REGION Network 24 (SCL): 5261/5263 SSC accumulator pressure LO/HI
   "DB_Alarms"."5261_SSC_PIT_01_Low".fLimit := 840.0;
   "DB_Alarms"."5261_SSC_PIT_01_Low".bEnable := TRUE;

   "DB_Alarms"."5263_SSC_PIT_01_High".fLimit := 1400.0;
   "DB_Alarms"."5263_SSC_PIT_01_High".bEnable := TRUE;
END_REGION

REGION Network 25 (SCL): 5262 SSC seal delta T HI
   "DB_Alarms"."5262_DeltaT_ShaftSealHigh".fLimit := 11.0;
   "DB_Alarms"."5262_DeltaT_ShaftSealHigh".bEnable := TRUE;
END_REGION
END_FUNCTION

FUNCTION_BLOCK "InputWarningHandling"   // FB7, FBD
TITLE = Handle I/O warnings
{ S7_Optimized_Access := 'TRUE' }
AUTHOR : Heaten
VERSION : 0.1
// stored: AutoNumber false, IsIECCheckEnabled false, IsRetainMemResEnabled false, MemoryReserve 100, SetENOAutomatically false, UDAEnableTagReadback false
   VAR
      A1101 { ExternalAccessible := 'False'; ExternalVisible := 'False'; ExternalWritable := 'False'; S7_SetPoint := 'True'} : "fbDigitalAlarm";
      A1121 { ExternalAccessible := 'False'; ExternalVisible := 'False'; ExternalWritable := 'False'; S7_SetPoint := 'True'} : "fbDigitalAlarm";
      A1140 { ExternalAccessible := 'False'; ExternalVisible := 'False'; ExternalWritable := 'False'; S7_SetPoint := 'True'} : "fbDigitalAlarm";
      A1216 { ExternalAccessible := 'False'; ExternalVisible := 'False'; ExternalWritable := 'False'; S7_SetPoint := 'True'} : "fbHMIEvent";
      A1217 { ExternalAccessible := 'False'; ExternalVisible := 'False'; ExternalWritable := 'False'; S7_SetPoint := 'True'} : "fbHMIEvent";
      A1218 { ExternalAccessible := 'False'; ExternalVisible := 'False'; ExternalWritable := 'False'; S7_SetPoint := 'True'} : "fbHMIEvent";
      A1224 { ExternalAccessible := 'False'; ExternalVisible := 'False'; ExternalWritable := 'False'; S7_SetPoint := 'True'} : "fbHMIEvent";
      A1225 { ExternalAccessible := 'False'; ExternalVisible := 'False'; ExternalWritable := 'False'; S7_SetPoint := 'True'} : "fbHMIEvent";
      A1226 { ExternalAccessible := 'False'; ExternalVisible := 'False'; ExternalWritable := 'False'; S7_SetPoint := 'True'} : "fbHMIEvent";
      A1227 { ExternalAccessible := 'False'; ExternalVisible := 'False'; ExternalWritable := 'False'; S7_SetPoint := 'True'} : "fbHMIEvent";
      A1228 { ExternalAccessible := 'False'; ExternalVisible := 'False'; ExternalWritable := 'False'; S7_SetPoint := 'True'} : "fbHMIEvent";
      A1229 { ExternalAccessible := 'False'; ExternalVisible := 'False'; ExternalWritable := 'False'; S7_SetPoint := 'True'} : "fbHMIEvent";
      A1230 { ExternalAccessible := 'False'; ExternalVisible := 'False'; ExternalWritable := 'False'; S7_SetPoint := 'True'} : "fbHMIEvent";
      A1234 { ExternalAccessible := 'False'; ExternalVisible := 'False'; ExternalWritable := 'False'; S7_SetPoint := 'True'} : "fbHMIEvent";
      A1235 { ExternalAccessible := 'False'; ExternalVisible := 'False'; ExternalWritable := 'False'; S7_SetPoint := 'True'} : "fbHMIEvent";
      A1236 { ExternalAccessible := 'False'; ExternalVisible := 'False'; ExternalWritable := 'False'; S7_SetPoint := 'True'} : "fbHMIEvent";
      A1237 { ExternalAccessible := 'False'; ExternalVisible := 'False'; ExternalWritable := 'False'; S7_SetPoint := 'True'} : "fbHMIEvent";
      A1238 { ExternalAccessible := 'False'; ExternalVisible := 'False'; ExternalWritable := 'False'; S7_SetPoint := 'True'} : "fbHMIEvent";
      A1239 { ExternalAccessible := 'False'; ExternalVisible := 'False'; ExternalWritable := 'False'; S7_SetPoint := 'True'} : "fbHMIEvent";
      A1240 { ExternalAccessible := 'False'; ExternalVisible := 'False'; ExternalWritable := 'False'; S7_SetPoint := 'True'} : "fbHMIEvent";
      A1245 { ExternalAccessible := 'False'; ExternalVisible := 'False'; ExternalWritable := 'False'; S7_SetPoint := 'True'} : "fbHMIEvent";
      A1246 { ExternalAccessible := 'False'; ExternalVisible := 'False'; ExternalWritable := 'False'; S7_SetPoint := 'True'} : "fbHMIEvent";
      A1247 { ExternalAccessible := 'False'; ExternalVisible := 'False'; ExternalWritable := 'False'; S7_SetPoint := 'True'} : "fbHMIEvent";
      A1248 { ExternalAccessible := 'False'; ExternalVisible := 'False'; ExternalWritable := 'False'; S7_SetPoint := 'True'} : "fbHMIEvent";
      A1249 { ExternalAccessible := 'False'; ExternalVisible := 'False'; ExternalWritable := 'False'; S7_SetPoint := 'True'} : "fbHMIEvent";
      A1251 { ExternalAccessible := 'False'; ExternalVisible := 'False'; ExternalWritable := 'False'; S7_SetPoint := 'True'} : "fbHMIEvent";
      A1252 { ExternalAccessible := 'False'; ExternalVisible := 'False'; ExternalWritable := 'False'; S7_SetPoint := 'True'} : "fbHMIEvent";
      A1253 { ExternalAccessible := 'False'; ExternalVisible := 'False'; ExternalWritable := 'False'; S7_SetPoint := 'True'} : "fbHMIEvent";
      A1254 { ExternalAccessible := 'False'; ExternalVisible := 'False'; ExternalWritable := 'False'; S7_SetPoint := 'True'} : "fbHMIEvent";
      A1258 { ExternalAccessible := 'False'; ExternalVisible := 'False'; ExternalWritable := 'False'; S7_SetPoint := 'True'} : "fbHMIEvent";
      A1259 { ExternalAccessible := 'False'; ExternalVisible := 'False'; ExternalWritable := 'False'; S7_SetPoint := 'True'} : "fbHMIEvent";
      A1260 { ExternalAccessible := 'False'; ExternalVisible := 'False'; ExternalWritable := 'False'; S7_SetPoint := 'True'} : "fbHMIEvent";
      A1262 { ExternalAccessible := 'False'; ExternalVisible := 'False'; ExternalWritable := 'False'; S7_SetPoint := 'True'} : "fbHMIEvent";
      A1263 { ExternalAccessible := 'False'; ExternalVisible := 'False'; ExternalWritable := 'False'; S7_SetPoint := 'True'} : "fbHMIEvent";
      A1265 { ExternalAccessible := 'False'; ExternalVisible := 'False'; ExternalWritable := 'False'; S7_SetPoint := 'True'} : "fbHMIEvent";
      A1269 { ExternalAccessible := 'False'; ExternalVisible := 'False'; ExternalWritable := 'False'; S7_SetPoint := 'True'} : "fbHMIEvent";
      A1270 { ExternalAccessible := 'False'; ExternalVisible := 'False'; ExternalWritable := 'False'; S7_SetPoint := 'True'} : "fbHMIEvent";
      A1271 { ExternalAccessible := 'False'; ExternalVisible := 'False'; ExternalWritable := 'False'; S7_SetPoint := 'True'} : "fbHMIEvent";
      A1272 { ExternalAccessible := 'False'; ExternalVisible := 'False'; ExternalWritable := 'False'; S7_SetPoint := 'True'} : "fbHMIEvent";
      A1273 { ExternalAccessible := 'False'; ExternalVisible := 'False'; ExternalWritable := 'False'; S7_SetPoint := 'True'} : "fbHMIEvent";
      A1275 { ExternalAccessible := 'False'; ExternalVisible := 'False'; ExternalWritable := 'False'; S7_SetPoint := 'True'} : "fbHMIEvent";
      A1293 { ExternalAccessible := 'False'; ExternalVisible := 'False'; ExternalWritable := 'False'; S7_SetPoint := 'True'} : "fbHMIEvent";
      A1294 { S7_SetPoint := 'True'} : "fbDigitalAlarm";
      A1295 { S7_SetPoint := 'True'} : "fbDigitalAlarm";
      A3401 { ExternalAccessible := 'False'; ExternalVisible := 'False'; ExternalWritable := 'False'; S7_SetPoint := 'True'} : "fbDigitalAlarm";
      A5200 { ExternalAccessible := 'False'; ExternalVisible := 'False'; ExternalWritable := 'False'; S7_SetPoint := 'True'} : "fbHMIEvent";
      A5201 { ExternalAccessible := 'False'; ExternalVisible := 'False'; ExternalWritable := 'False'; S7_SetPoint := 'True'} : "fbHMIEvent";
      A5202 { ExternalAccessible := 'False'; ExternalVisible := 'False'; ExternalWritable := 'False'; S7_SetPoint := 'True'} : "fbHMIEvent";
      A5203 { ExternalAccessible := 'False'; ExternalVisible := 'False'; ExternalWritable := 'False'; S7_SetPoint := 'True'} : "fbDigitalAlarm";
      A5204 { ExternalAccessible := 'False'; ExternalVisible := 'False'; ExternalWritable := 'False'; S7_SetPoint := 'True'} : "fbDigitalAlarm";
      A5206 { ExternalAccessible := 'False'; ExternalVisible := 'False'; ExternalWritable := 'False'; S7_SetPoint := 'True'} : "fbHMIEvent";
      A5256 { ExternalAccessible := 'False'; ExternalVisible := 'False'; ExternalWritable := 'False'; S7_SetPoint := 'True'} : "fbHMIEvent";
   END_VAR
BEGIN

REGION Network 1: 1101
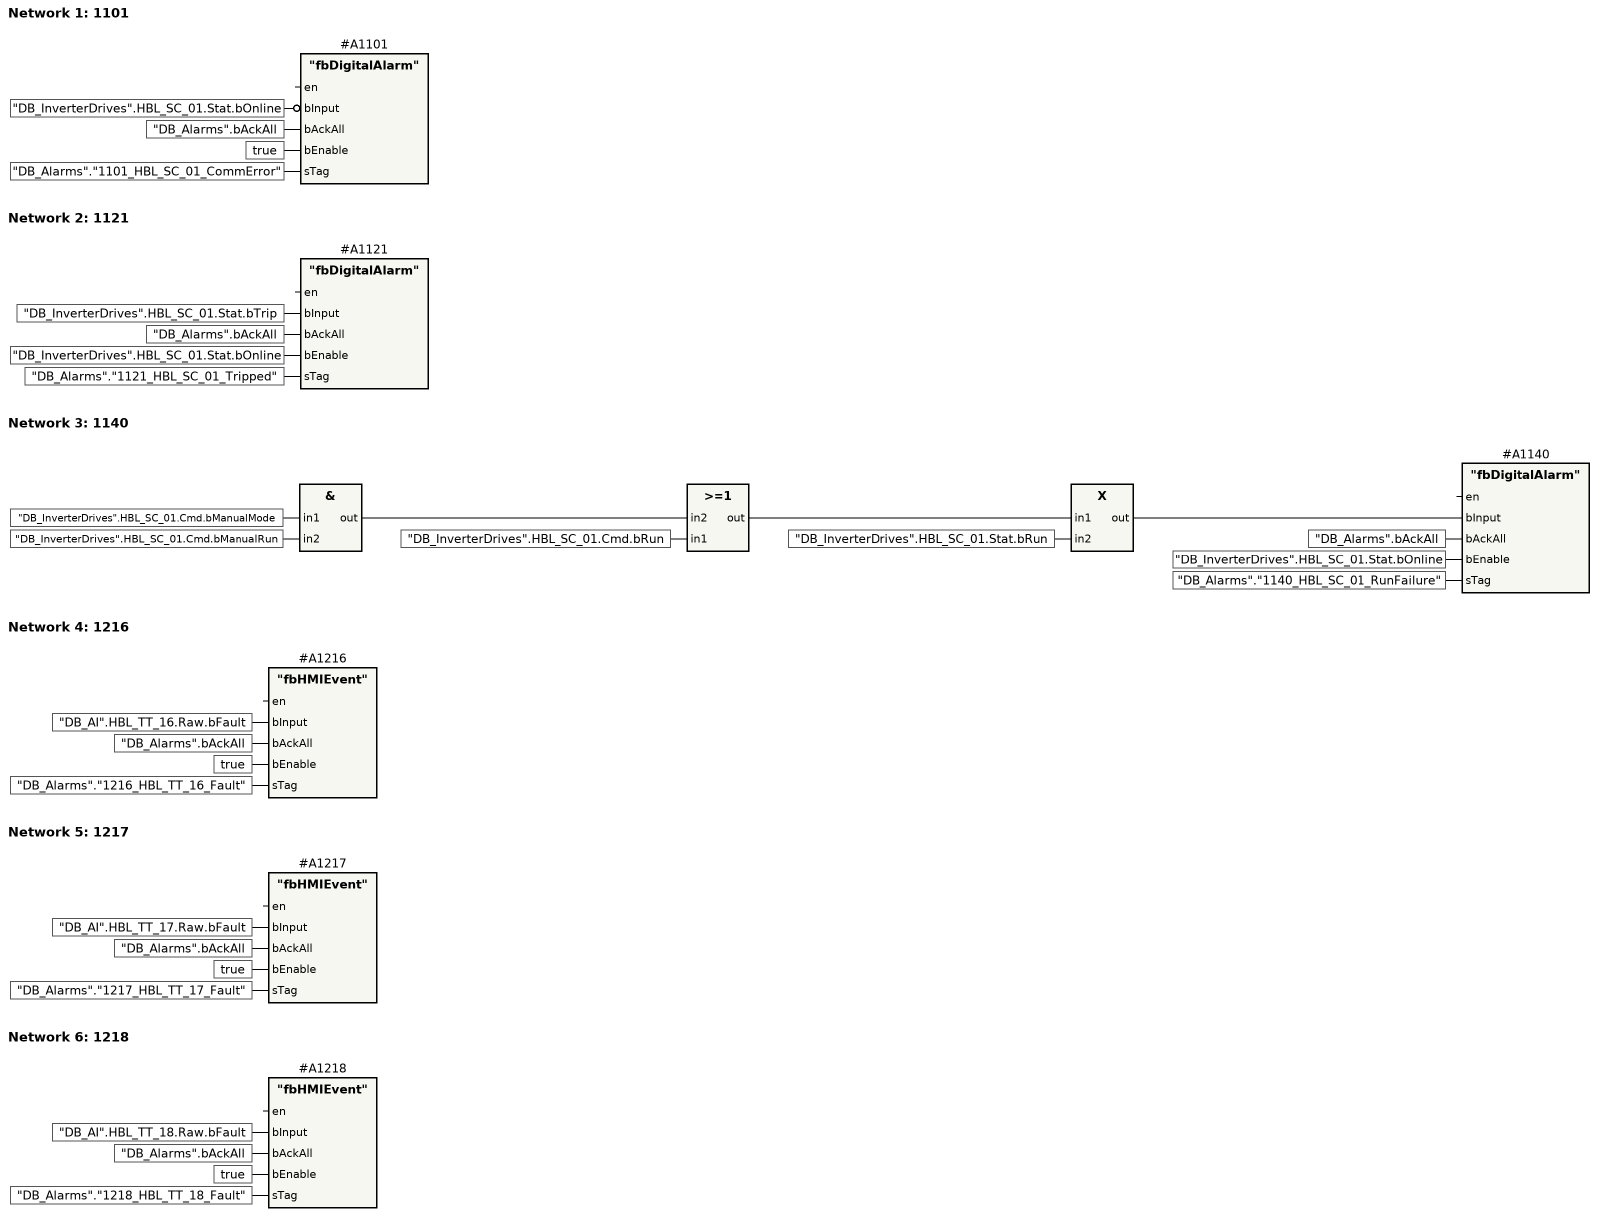
   #A1101(bInput := NOT "DB_InverterDrives".HBL_SC_01.Stat.bOnline,   // "fbDigitalAlarm"
          bAckAll := "DB_Alarms".bAckAll,
          bEnable := true,
          sTag := "DB_Alarms"."1101_HBL_SC_01_CommError");
END_REGION

REGION Network 2: 1121
   #A1121(bInput := "DB_InverterDrives".HBL_SC_01.Stat.bTrip,   // "fbDigitalAlarm"
          bAckAll := "DB_Alarms".bAckAll,
          bEnable := "DB_InverterDrives".HBL_SC_01.Stat.bOnline,
          sTag := "DB_Alarms"."1121_HBL_SC_01_Tripped");
END_REGION

REGION Network 3: 1140
   #A1140(bInput := (("DB_InverterDrives".HBL_SC_01.Cmd.bManualMode AND "DB_InverterDrives".HBL_SC_01.Cmd.bManualRun) OR "DB_InverterDrives".HBL_SC_01.Cmd.bRun) XOR "DB_InverterDrives".HBL_SC_01.Stat.bRun,   // "fbDigitalAlarm"
          bAckAll := "DB_Alarms".bAckAll,
          bEnable := "DB_InverterDrives".HBL_SC_01.Stat.bOnline,
          sTag := "DB_Alarms"."1140_HBL_SC_01_RunFailure");
END_REGION

REGION Network 4: 1216
   #A1216(bInput := "DB_AI".HBL_TT_16.Raw.bFault,   // "fbHMIEvent"
          bAckAll := "DB_Alarms".bAckAll,
          bEnable := true,
          sTag := "DB_Alarms"."1216_HBL_TT_16_Fault");
END_REGION

REGION Network 5: 1217
   #A1217(bInput := "DB_AI".HBL_TT_17.Raw.bFault,   // "fbHMIEvent"
          bAckAll := "DB_Alarms".bAckAll,
          bEnable := true,
          sTag := "DB_Alarms"."1217_HBL_TT_17_Fault");
END_REGION

REGION Network 6: 1218
   #A1218(bInput := "DB_AI".HBL_TT_18.Raw.bFault,   // "fbHMIEvent"
          bAckAll := "DB_Alarms".bAckAll,
          bEnable := true,
          sTag := "DB_Alarms"."1218_HBL_TT_18_Fault");
END_REGION

REGION Network 7: 1224
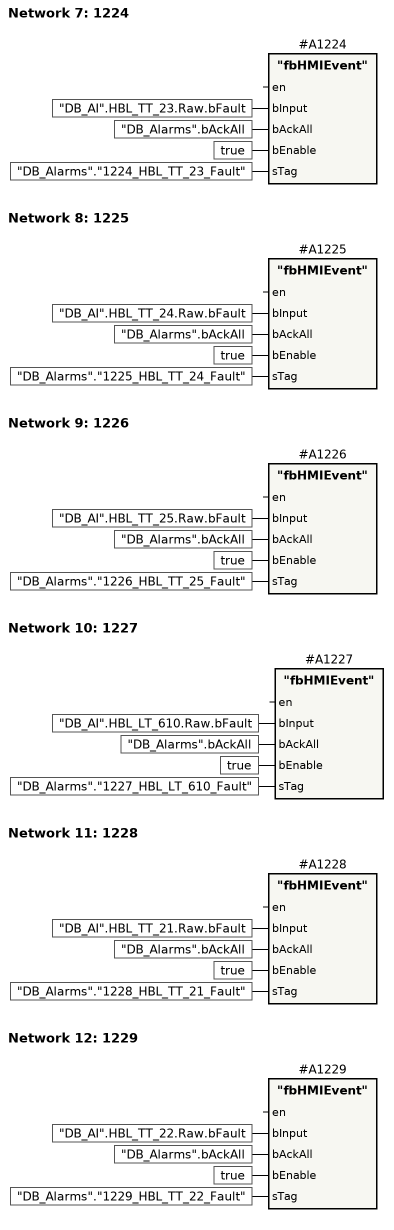
   #A1224(bInput := "DB_AI".HBL_TT_23.Raw.bFault,   // "fbHMIEvent"
          bAckAll := "DB_Alarms".bAckAll,
          bEnable := true,
          sTag := "DB_Alarms"."1224_HBL_TT_23_Fault");
END_REGION

REGION Network 8: 1225
   #A1225(bInput := "DB_AI".HBL_TT_24.Raw.bFault,   // "fbHMIEvent"
          bAckAll := "DB_Alarms".bAckAll,
          bEnable := true,
          sTag := "DB_Alarms"."1225_HBL_TT_24_Fault");
END_REGION

REGION Network 9: 1226
   #A1226(bInput := "DB_AI".HBL_TT_25.Raw.bFault,   // "fbHMIEvent"
          bAckAll := "DB_Alarms".bAckAll,
          bEnable := true,
          sTag := "DB_Alarms"."1226_HBL_TT_25_Fault");
END_REGION

REGION Network 10: 1227
   #A1227(bInput := "DB_AI".HBL_LT_610.Raw.bFault,   // "fbHMIEvent"
          bAckAll := "DB_Alarms".bAckAll,
          bEnable := true,
          sTag := "DB_Alarms"."1227_HBL_LT_610_Fault");
END_REGION

REGION Network 11: 1228
   #A1228(bInput := "DB_AI".HBL_TT_21.Raw.bFault,   // "fbHMIEvent"
          bAckAll := "DB_Alarms".bAckAll,
          bEnable := true,
          sTag := "DB_Alarms"."1228_HBL_TT_21_Fault");
END_REGION

REGION Network 12: 1229
   #A1229(bInput := "DB_AI".HBL_TT_22.Raw.bFault,   // "fbHMIEvent"
          bAckAll := "DB_Alarms".bAckAll,
          bEnable := true,
          sTag := "DB_Alarms"."1229_HBL_TT_22_Fault");
END_REGION

REGION Network 13: 1230
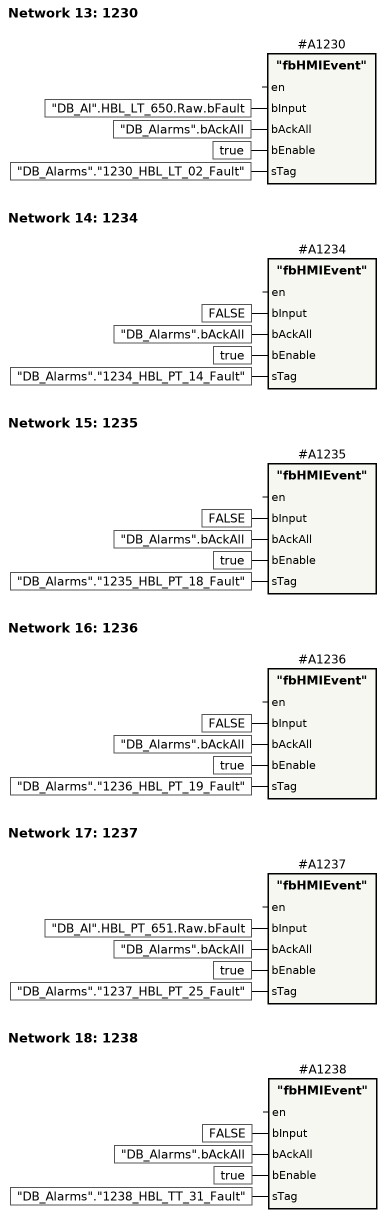
   #A1230(bInput := "DB_AI".HBL_LT_650.Raw.bFault,   // "fbHMIEvent"
          bAckAll := "DB_Alarms".bAckAll,
          bEnable := true,
          sTag := "DB_Alarms"."1230_HBL_LT_02_Fault");
END_REGION

REGION Network 14: 1234
   #A1234(bInput := FALSE,   // "fbHMIEvent"
          bAckAll := "DB_Alarms".bAckAll,
          bEnable := true,
          sTag := "DB_Alarms"."1234_HBL_PT_14_Fault");
END_REGION

REGION Network 15: 1235
   #A1235(bInput := FALSE,   // "fbHMIEvent"
          bAckAll := "DB_Alarms".bAckAll,
          bEnable := true,
          sTag := "DB_Alarms"."1235_HBL_PT_18_Fault");
END_REGION

REGION Network 16: 1236
   #A1236(bInput := FALSE,   // "fbHMIEvent"
          bAckAll := "DB_Alarms".bAckAll,
          bEnable := true,
          sTag := "DB_Alarms"."1236_HBL_PT_19_Fault");
END_REGION

REGION Network 17: 1237
   #A1237(bInput := "DB_AI".HBL_PT_651.Raw.bFault,   // "fbHMIEvent"
          bAckAll := "DB_Alarms".bAckAll,
          bEnable := true,
          sTag := "DB_Alarms"."1237_HBL_PT_25_Fault");
END_REGION

REGION Network 18: 1238
   #A1238(bInput := FALSE,   // "fbHMIEvent"
          bAckAll := "DB_Alarms".bAckAll,
          bEnable := true,
          sTag := "DB_Alarms"."1238_HBL_TT_31_Fault");
END_REGION

REGION Network 19: 1239
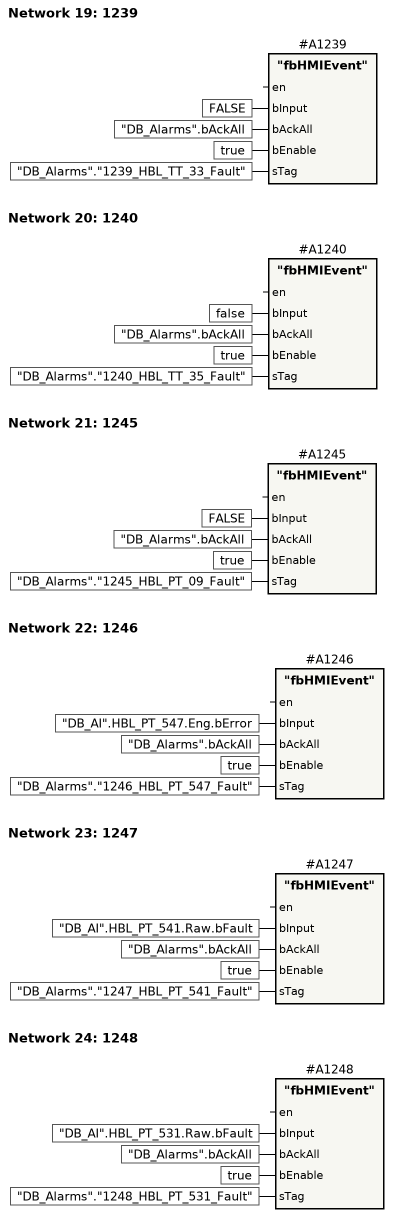
   #A1239(bInput := FALSE,   // "fbHMIEvent"
          bAckAll := "DB_Alarms".bAckAll,
          bEnable := true,
          sTag := "DB_Alarms"."1239_HBL_TT_33_Fault");
END_REGION

REGION Network 20: 1240
   #A1240(bInput := false,   // "fbHMIEvent"
          bAckAll := "DB_Alarms".bAckAll,
          bEnable := true,
          sTag := "DB_Alarms"."1240_HBL_TT_35_Fault");
END_REGION

REGION Network 21: 1245
   #A1245(bInput := FALSE,   // "fbHMIEvent"
          bAckAll := "DB_Alarms".bAckAll,
          bEnable := true,
          sTag := "DB_Alarms"."1245_HBL_PT_09_Fault");
END_REGION

REGION Network 22: 1246
   #A1246(bInput := "DB_AI".HBL_PT_547.Eng.bError,   // "fbHMIEvent"
          bAckAll := "DB_Alarms".bAckAll,
          bEnable := true,
          sTag := "DB_Alarms"."1246_HBL_PT_547_Fault");
END_REGION

REGION Network 23: 1247
   #A1247(bInput := "DB_AI".HBL_PT_541.Raw.bFault,   // "fbHMIEvent"
          bAckAll := "DB_Alarms".bAckAll,
          bEnable := true,
          sTag := "DB_Alarms"."1247_HBL_PT_541_Fault");
END_REGION

REGION Network 24: 1248
   #A1248(bInput := "DB_AI".HBL_PT_531.Raw.bFault,   // "fbHMIEvent"
          bAckAll := "DB_Alarms".bAckAll,
          bEnable := true,
          sTag := "DB_Alarms"."1248_HBL_PT_531_Fault");
END_REGION

REGION Network 25: 1249
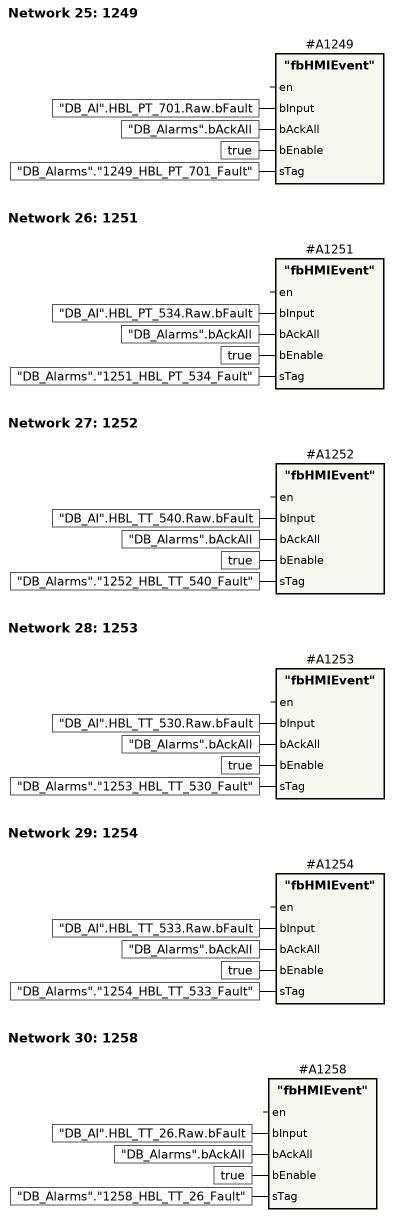
   #A1249(bInput := "DB_AI".HBL_PT_701.Raw.bFault,   // "fbHMIEvent"
          bAckAll := "DB_Alarms".bAckAll,
          bEnable := true,
          sTag := "DB_Alarms"."1249_HBL_PT_701_Fault");
END_REGION

REGION Network 26: 1251
   #A1251(bInput := "DB_AI".HBL_PT_534.Raw.bFault,   // "fbHMIEvent"
          bAckAll := "DB_Alarms".bAckAll,
          bEnable := true,
          sTag := "DB_Alarms"."1251_HBL_PT_534_Fault");
END_REGION

REGION Network 27: 1252
   #A1252(bInput := "DB_AI".HBL_TT_540.Raw.bFault,   // "fbHMIEvent"
          bAckAll := "DB_Alarms".bAckAll,
          bEnable := true,
          sTag := "DB_Alarms"."1252_HBL_TT_540_Fault");
END_REGION

REGION Network 28: 1253
   #A1253(bInput := "DB_AI".HBL_TT_530.Raw.bFault,   // "fbHMIEvent"
          bAckAll := "DB_Alarms".bAckAll,
          bEnable := true,
          sTag := "DB_Alarms"."1253_HBL_TT_530_Fault");
END_REGION

REGION Network 29: 1254
   #A1254(bInput := "DB_AI".HBL_TT_533.Raw.bFault,   // "fbHMIEvent"
          bAckAll := "DB_Alarms".bAckAll,
          bEnable := true,
          sTag := "DB_Alarms"."1254_HBL_TT_533_Fault");
END_REGION

REGION Network 30: 1258
   #A1258(bInput := "DB_AI".HBL_TT_26.Raw.bFault,   // "fbHMIEvent"
          bAckAll := "DB_Alarms".bAckAll,
          bEnable := true,
          sTag := "DB_Alarms"."1258_HBL_TT_26_Fault");
END_REGION

REGION Network 31: 1259
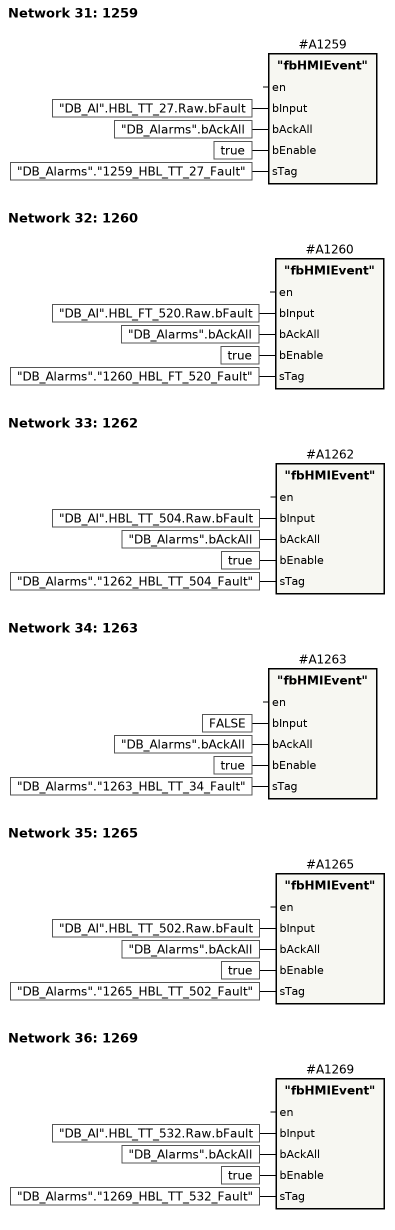
   #A1259(bInput := "DB_AI".HBL_TT_27.Raw.bFault,   // "fbHMIEvent"
          bAckAll := "DB_Alarms".bAckAll,
          bEnable := true,
          sTag := "DB_Alarms"."1259_HBL_TT_27_Fault");
END_REGION

REGION Network 32: 1260
   #A1260(bInput := "DB_AI".HBL_FT_520.Raw.bFault,   // "fbHMIEvent"
          bAckAll := "DB_Alarms".bAckAll,
          bEnable := true,
          sTag := "DB_Alarms"."1260_HBL_FT_520_Fault");
END_REGION

REGION Network 33: 1262
   #A1262(bInput := "DB_AI".HBL_TT_504.Raw.bFault,   // "fbHMIEvent"
          bAckAll := "DB_Alarms".bAckAll,
          bEnable := true,
          sTag := "DB_Alarms"."1262_HBL_TT_504_Fault");
END_REGION

REGION Network 34: 1263
   #A1263(bInput := FALSE,   // "fbHMIEvent"
          bAckAll := "DB_Alarms".bAckAll,
          bEnable := true,
          sTag := "DB_Alarms"."1263_HBL_TT_34_Fault");
END_REGION

REGION Network 35: 1265
   #A1265(bInput := "DB_AI".HBL_TT_502.Raw.bFault,   // "fbHMIEvent"
          bAckAll := "DB_Alarms".bAckAll,
          bEnable := true,
          sTag := "DB_Alarms"."1265_HBL_TT_502_Fault");
END_REGION

REGION Network 36: 1269
   #A1269(bInput := "DB_AI".HBL_TT_532.Raw.bFault,   // "fbHMIEvent"
          bAckAll := "DB_Alarms".bAckAll,
          bEnable := true,
          sTag := "DB_Alarms"."1269_HBL_TT_532_Fault");
END_REGION

REGION Network 37: 1270
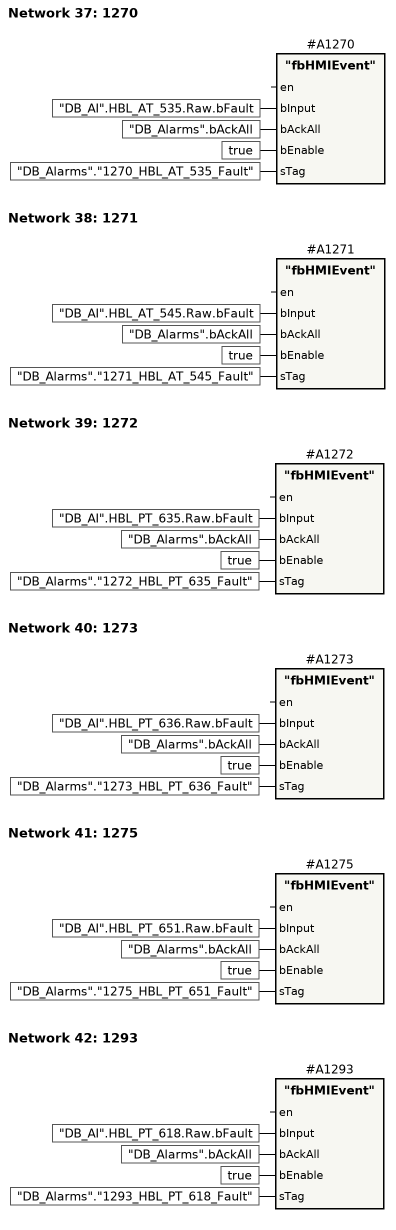
   #A1270(bInput := "DB_AI".HBL_AT_535.Raw.bFault,   // "fbHMIEvent"
          bAckAll := "DB_Alarms".bAckAll,
          bEnable := true,
          sTag := "DB_Alarms"."1270_HBL_AT_535_Fault");
END_REGION

REGION Network 38: 1271
   #A1271(bInput := "DB_AI".HBL_AT_545.Raw.bFault,   // "fbHMIEvent"
          bAckAll := "DB_Alarms".bAckAll,
          bEnable := true,
          sTag := "DB_Alarms"."1271_HBL_AT_545_Fault");
END_REGION

REGION Network 39: 1272
   #A1272(bInput := "DB_AI".HBL_PT_635.Raw.bFault,   // "fbHMIEvent"
          bAckAll := "DB_Alarms".bAckAll,
          bEnable := true,
          sTag := "DB_Alarms"."1272_HBL_PT_635_Fault");
END_REGION

REGION Network 40: 1273
   #A1273(bInput := "DB_AI".HBL_PT_636.Raw.bFault,   // "fbHMIEvent"
          bAckAll := "DB_Alarms".bAckAll,
          bEnable := true,
          sTag := "DB_Alarms"."1273_HBL_PT_636_Fault");
END_REGION

REGION Network 41: 1275
   #A1275(bInput := "DB_AI".HBL_PT_651.Raw.bFault,   // "fbHMIEvent"
          bAckAll := "DB_Alarms".bAckAll,
          bEnable := true,
          sTag := "DB_Alarms"."1275_HBL_PT_651_Fault");
END_REGION

REGION Network 42: 1293
   #A1293(bInput := "DB_AI".HBL_PT_618.Raw.bFault,   // "fbHMIEvent"
          bAckAll := "DB_Alarms".bAckAll,
          bEnable := true,
          sTag := "DB_Alarms"."1293_HBL_PT_618_Fault");
END_REGION

REGION Network 43: 1294
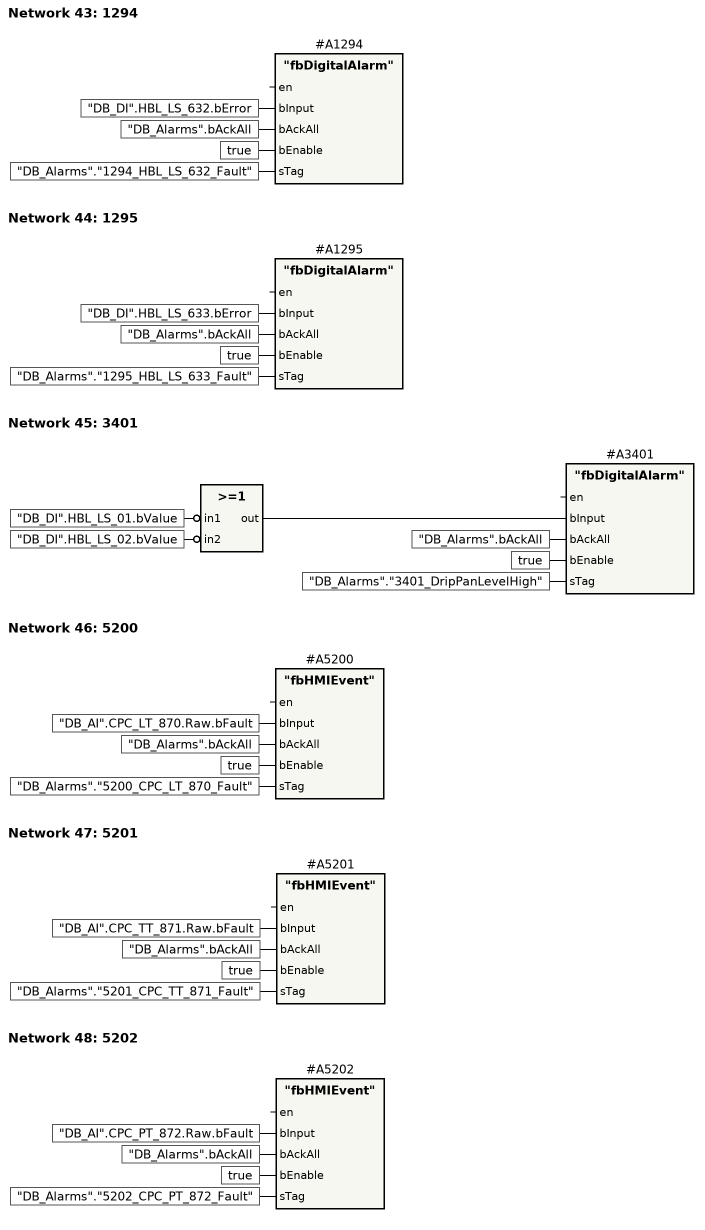
   #A1294(bInput := "DB_DI".HBL_LS_632.bError,   // "fbDigitalAlarm"
          bAckAll := "DB_Alarms".bAckAll,
          bEnable := true,
          sTag := "DB_Alarms"."1294_HBL_LS_632_Fault");
END_REGION

REGION Network 44: 1295
   #A1295(bInput := "DB_DI".HBL_LS_633.bError,   // "fbDigitalAlarm"
          bAckAll := "DB_Alarms".bAckAll,
          bEnable := true,
          sTag := "DB_Alarms"."1295_HBL_LS_633_Fault");
END_REGION

REGION Network 45: 3401
   #A3401(bInput := NOT "DB_DI".HBL_LS_01.bValue OR NOT "DB_DI".HBL_LS_02.bValue,   // "fbDigitalAlarm"
          bAckAll := "DB_Alarms".bAckAll,
          bEnable := true,
          sTag := "DB_Alarms"."3401_DripPanLevelHigh");
END_REGION

REGION Network 46: 5200
   #A5200(bInput := "DB_AI".CPC_LT_870.Raw.bFault,   // "fbHMIEvent"
          bAckAll := "DB_Alarms".bAckAll,
          bEnable := true,
          sTag := "DB_Alarms"."5200_CPC_LT_870_Fault");
END_REGION

REGION Network 47: 5201
   #A5201(bInput := "DB_AI".CPC_TT_871.Raw.bFault,   // "fbHMIEvent"
          bAckAll := "DB_Alarms".bAckAll,
          bEnable := true,
          sTag := "DB_Alarms"."5201_CPC_TT_871_Fault");
END_REGION

REGION Network 48: 5202
   #A5202(bInput := "DB_AI".CPC_PT_872.Raw.bFault,   // "fbHMIEvent"
          bAckAll := "DB_Alarms".bAckAll,
          bEnable := true,
          sTag := "DB_Alarms"."5202_CPC_PT_872_Fault");
END_REGION

REGION Network 49: 5203
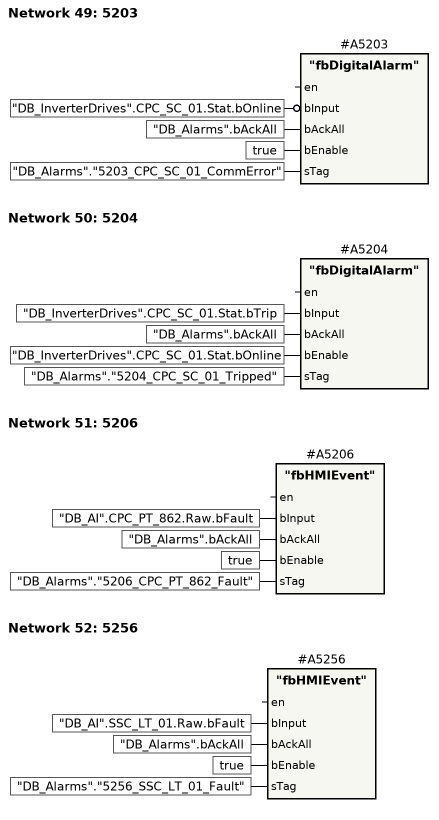
   #A5203(bInput := NOT "DB_InverterDrives".CPC_SC_01.Stat.bOnline,   // "fbDigitalAlarm"
          bAckAll := "DB_Alarms".bAckAll,
          bEnable := true,
          sTag := "DB_Alarms"."5203_CPC_SC_01_CommError");
END_REGION

REGION Network 50: 5204
   // Only show if online
   #A5204(bInput := "DB_InverterDrives".CPC_SC_01.Stat.bTrip,   // "fbDigitalAlarm"
          bAckAll := "DB_Alarms".bAckAll,
          bEnable := "DB_InverterDrives".CPC_SC_01.Stat.bOnline,
          sTag := "DB_Alarms"."5204_CPC_SC_01_Tripped");
END_REGION

REGION Network 51: 5206
   #A5206(bInput := "DB_AI".CPC_PT_862.Raw.bFault,   // "fbHMIEvent"
          bAckAll := "DB_Alarms".bAckAll,
          bEnable := true,
          sTag := "DB_Alarms"."5206_CPC_PT_862_Fault");
END_REGION

REGION Network 52: 5256
   #A5256(bInput := "DB_AI".SSC_LT_01.Raw.bFault,   // "fbHMIEvent"
          bAckAll := "DB_Alarms".bAckAll,
          bEnable := true,
          sTag := "DB_Alarms"."5256_SSC_LT_01_Fault");
END_REGION
END_FUNCTION_BLOCK

FUNCTION_BLOCK "fbDigitalAlarm"   // FB47, FBD
{ S7_Optimized_Access := 'TRUE' }
VERSION : 0.1
// stored: AutoNumber true, IsIECCheckEnabled false, IsRetainMemResEnabled false, MemoryReserve 0, SetENOAutomatically false, UDAEnableTagReadback false
   VAR_INPUT
      bInput : Bool;
      bAckAll : Bool;
      bEnable : Bool;
   END_VAR
   VAR_IN_OUT
      sTag : "stDigitalAlarm";
   END_VAR
   VAR
      Alarm : "fbAlarm";
   END_VAR
BEGIN

REGION Network 1
   // The Enables are ANDed together to allow the struct one to act as a disable bit
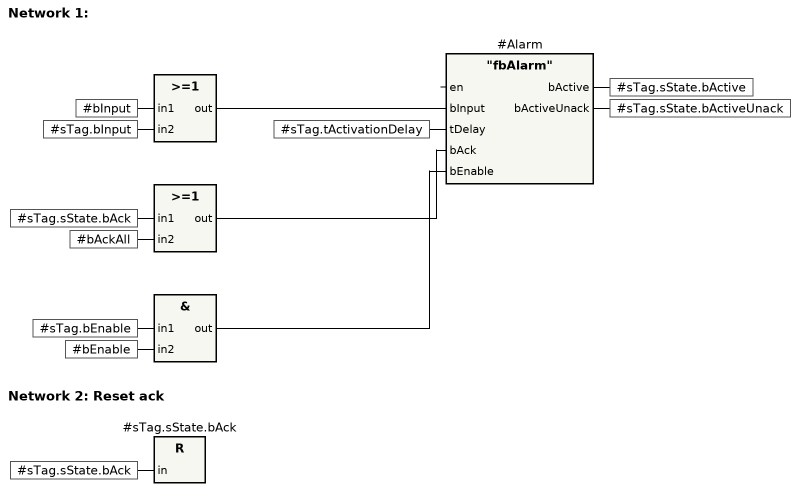
   #Alarm(bInput := #bInput OR #sTag.bInput,   // "fbAlarm"
          tDelay := #sTag.tActivationDelay,
          bAck := #sTag.sState.bAck OR #bAckAll,
          bEnable := #sTag.bEnable AND #bEnable,
          bActive => #sTag.sState.bActive,
          bActiveUnack => #sTag.sState.bActiveUnack);
END_REGION

REGION Network 2: Reset ack
   IF #sTag.sState.bAck THEN #sTag.sState.bAck := FALSE; END_IF;
END_REGION
END_FUNCTION_BLOCK

FUNCTION_BLOCK "fbAlarm"   // FB40, FBD
TITLE = Alarm with time delay
{ S7_Optimized_Access := 'TRUE' }
VERSION : 0.1
// stored: AutoNumber true, IsIECCheckEnabled false, IsRetainMemResEnabled false, MemoryReserve 0, SetENOAutomatically false, UDAEnableTagReadback false
   VAR_INPUT
      bInput : Bool;
      tDelay : Time;
      bAck : Bool;
      bEnable : Bool;
   END_VAR
   VAR_OUTPUT
      bActive : Bool;
      bActiveUnack : Bool;
   END_VAR
   VAR
      DelayTimer : TON_TIME;
      Alarm : Bool;
      AlarmUnack : Bool;
      mActive : Bool;
   END_VAR
   VAR_TEMP
      DelayExpired : Bool;
   END_VAR
   VAR_TEMP   // added for the SCL form of the ladder/FBD networks
      _w1 : Bool;
   END_VAR
BEGIN

REGION Network 1: Delay: alarm must be active for a minimum time period
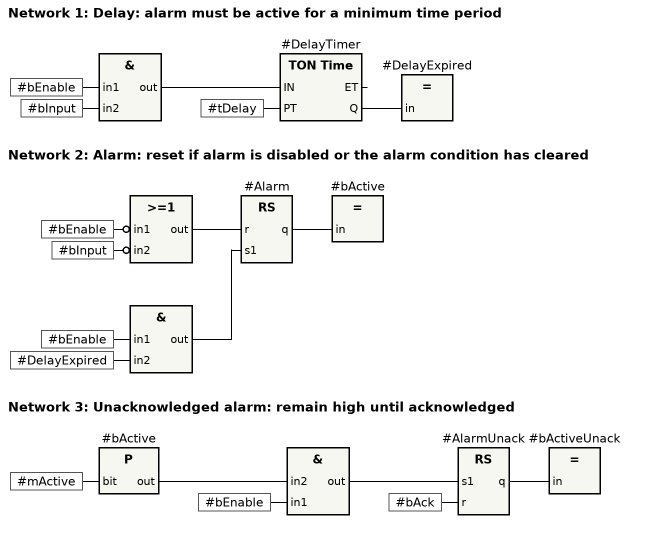
   #DelayTimer(IN := #bEnable AND #bInput, PT := #tDelay);   // TON
   #DelayExpired := #DelayTimer.Q;
END_REGION

REGION Network 2: Alarm: reset if alarm is disabled or the alarm condition has cleared
   IF NOT #bEnable OR NOT #bInput THEN
       #Alarm := FALSE;   // RS flip-flop
   END_IF;
   IF #bEnable AND #DelayExpired THEN #Alarm := TRUE; END_IF;
   #bActive := #Alarm;
END_REGION

REGION Network 3: Unacknowledged alarm: remain high until acknowledged
   #_w1 := #bActive AND NOT #mActive;   // rising edge of #bActive
   #mActive := #bActive;
   IF #bAck THEN
       #AlarmUnack := FALSE;   // RS flip-flop
   END_IF;
   IF #_w1 AND #bEnable THEN #AlarmUnack := TRUE; END_IF;
   #bActiveUnack := #AlarmUnack;
END_REGION
END_FUNCTION_BLOCK

FUNCTION_BLOCK "HMI-Communication"   // FB3, FBD
{ S7_Optimized_Access := 'TRUE' }
VERSION : 0.1
// stored: AutoNumber true, IsIECCheckEnabled false, IsRetainMemResEnabled false, MemoryReserve 0, SetENOAutomatically false, UDAEnableTagReadback false
   VAR
      StartRequest : Bool;
      StopRequest : Bool;
      HMI_Running : Bool;
      SkipPauseTime : Bool;
      EmergencyStopWaitTime : Bool;
      SkipEmergencyStopWait : Bool;
      CloseSafetyRelay : Bool;
      OpenSafetyRelay : Bool;
      HMI_Acknowledge_Error : Bool;
      BackToStandby_OilHeat { ExternalVisible := 'False'; ExternalWritable := 'False'} : Bool;
      BackToStandby_SourceFlowNotOK { ExternalVisible := 'False'; ExternalWritable := 'False'} : Bool;
      BackToStandby_SinkFlowNotOK : Bool;
      BackToStandby_SinkTemperatureNotOK : Bool;
      BackToStandby_SourceTemperatureNotOK : Bool;
      BackToStandby_PerformanceControlNotOK : Bool;
      ReturnValvesManualOverride : Bool;   // Hopefully temporary!
      HBL_XV_02override : Bool;   // Temporary!
      HBL_XV_03override : Bool;   // Temporary!
      HBL_HV_860override : Bool;   // Temporary!
      HBL_HV_861override : Bool;   // Temporary!
      State_Text : String;
      BackToStandby_TriggerBit : Bool;   // Bit set if state changes "back to standby"
      BackToStandby_TriggerMemory : Bool;   // Internal flag memory for "back to standby" changes
      BackToStandby_TriggerInt : Int;   // Integer for state changes "back to standby" HMI message
      BackToStandbyReason_Text : String;   // Text to describe "back to standby" reason
      StopReason_TriggerBit : Bool;
      StopReason_TriggerMemory : Bool;
      StopReason_TriggerInt : Int;
      StopReason_Text : String;
      Progress_Text : Int;
      RegulationTarget : Int;
      RegulationTargetPrev : Int;
      HeatboosterSetpoint : Real;   // Main setpoint of the machine
      HeatboosterSetpointPrev : Real;
      EmergencyStopCountdown : Time_Of_Day;
      A1001 { ExternalAccessible := 'False'; ExternalVisible := 'False'; ExternalWritable := 'False'} : "fbHMIEvent";
      WinCCLink { ExternalAccessible := 'False'; ExternalVisible := 'False'; ExternalWritable := 'False'; S7_SetPoint := 'True'} : "fbHeartbeat";
      State2DwellTimeElapsed { S7_SetPoint := 'True'} : Time_Of_Day;
      State2DwellTime : Time_Of_Day;
      State3DwellTimeElapsed : Time_Of_Day;
      State3DwellTime : Time_Of_Day;
      State4DwellTimeElapsed : Time_Of_Day;
      State4DwellTime : Time_Of_Day;
      State5DwellTimeElapsed : Time_Of_Day;
      State5DwellTime : Time_Of_Day;
      State7DwellTimeElapsed : Time_Of_Day;
      State7DwellTime : Time_Of_Day;
      State2PauseTimeElapsed : Time_Of_Day;
      State2PauseTime : Time_Of_Day;
      PurgeControlPurgeTime : Time_Of_Day;
      PurgeControlSpinTime : Time_Of_Day;
      PerformanceControlStandbyTime : Time_Of_Day;
      PerformanceControlStandbyTimeElapsed : Time_Of_Day;
      FilterDryerOnTime : Time_Of_Day;
      FilterDryerOffTime : Time_Of_Day;
      OilRecoveryOnTime : Time_Of_Day;
      ProgressiveTimes : Array[0..3] of Time_Of_Day;
      ProgressiveTime : Time_Of_Day;
      ProgressiveManualTime : Time_Of_Day;
      HV640_OpenTime : Time_Of_Day;
      HV640_CloseTime : Time_Of_Day;
      HV670_OpenTime : Time_Of_Day;
      HV670_CloseTime : Time_Of_Day;
      HV852_OpenTime : Time_Of_Day;
      HV852_CloseTime : Time_Of_Day;
      HV861_OpenTime : Time_Of_Day;
      HV861_CloseTime : Time_Of_Day;
      State2DwellSync { ExternalAccessible := 'False'; ExternalVisible := 'False'; ExternalWritable := 'False'} : "fbWinCCTime";
      State3DwellSync { ExternalAccessible := 'False'; ExternalVisible := 'False'; ExternalWritable := 'False'; S7_SetPoint := 'True'} : "fbWinCCTime";
      State4DwellSync { ExternalAccessible := 'False'; ExternalVisible := 'False'; ExternalWritable := 'False'; S7_SetPoint := 'True'} : "fbWinCCTime";
      State5DwellSync { ExternalAccessible := 'False'; ExternalVisible := 'False'; ExternalWritable := 'False'; S7_SetPoint := 'True'} : "fbWinCCTime";
      State7DwellSync { ExternalAccessible := 'False'; ExternalVisible := 'False'; ExternalWritable := 'False'; S7_SetPoint := 'True'} : "fbWinCCTime";
      State2PauseSync { ExternalAccessible := 'False'; ExternalVisible := 'False'; ExternalWritable := 'False'; S7_SetPoint := 'True'} : "fbWinCCTime";
      PurgeControlPurgeSync { ExternalAccessible := 'False'; ExternalVisible := 'False'; ExternalWritable := 'False'; S7_SetPoint := 'True'} : "fbWinCCTime";
      PurgeControlSpinSync { ExternalAccessible := 'False'; ExternalVisible := 'False'; ExternalWritable := 'False'; S7_SetPoint := 'True'} : "fbWinCCTime";
      ProgressiveTime0Sync { ExternalAccessible := 'False'; ExternalVisible := 'False'; ExternalWritable := 'False'; S7_SetPoint := 'True'} : "fbWinCCTime";
      ProgressiveTime1Sync { ExternalAccessible := 'False'; ExternalVisible := 'False'; ExternalWritable := 'False'; S7_SetPoint := 'True'} : "fbWinCCTime";
      ProgressiveTime2Sync { ExternalAccessible := 'False'; ExternalVisible := 'False'; ExternalWritable := 'False'; S7_SetPoint := 'True'} : "fbWinCCTime";
      ProgressiveTime3Sync { ExternalAccessible := 'False'; ExternalVisible := 'False'; ExternalWritable := 'False'; S7_SetPoint := 'True'} : "fbWinCCTime";
      ProgressiveManualTimeSync { ExternalAccessible := 'False'; ExternalVisible := 'False'; ExternalWritable := 'False'; S7_SetPoint := 'True'} : "fbWinCCTime";
      PerformanceControlStandbySync { ExternalAccessible := 'False'; ExternalVisible := 'False'; ExternalWritable := 'False'; S7_SetPoint := 'True'} : "fbWinCCTime";
      FilterDryerOnTimeSync { S7_SetPoint := 'True'} : "fbWinCCTime";
      FilterDryerOffTimeSync { S7_SetPoint := 'True'} : "fbWinCCTime";
      OilRecoveryOnTimeSync { S7_SetPoint := 'True'} : "fbWinCCTime";
      HV640_OpenTimeSync { S7_SetPoint := 'True'} : "fbWinCCTime";
      HV640_CloseTimeSync { S7_SetPoint := 'True'} : "fbWinCCTime";
      HV670_OpenTimeSync { S7_SetPoint := 'True'} : "fbWinCCTime";
      HV670_CloseTimeSync { S7_SetPoint := 'True'} : "fbWinCCTime";
      HV852_OpenTimeSync { S7_SetPoint := 'True'} : "fbWinCCTime";
      HV852_CloseTimeSync { S7_SetPoint := 'True'} : "fbWinCCTime";
      HV861_OpenTimeSync { S7_SetPoint := 'True'} : "fbWinCCTime";
      HV861_CloseTimeSync { S7_SetPoint := 'True'} : "fbWinCCTime";
   END_VAR
   VAR_TEMP
      FellBackToStandby_456 : Bool;
      FellBackToStandby_56 : Bool;
   END_VAR
   VAR CONSTANT
      "01_WaitingForStateChange" : SInt := 1;
      "02_ErrorAcknowledge" : SInt := 2;
      "03_SafetyRelayNotClosed" : SInt := 3;
      "04_SafetyRelayInterrupted" : SInt := 4;
      "05_CPU_Init" : SInt := 5;
      "6_CriticalAlarmActive" : SInt := 6;
      "10_ReadyToStart" : SInt := 10;
      "11_EmergencyStopActive" : SInt := 11;
      "12_InverterNotOnline" : SInt := 12;
      "13_ReadyToStartWithActiveWarnings" : SInt := 13;
      "14_EmergencyStopWaitTime" : SInt := 14;
      "20_WaitForSourceFlow" : SInt := 20;
      "21_WaitForSinkFlow" : SInt := 21;
      "22_WaitForSinkHeat" : SInt := 22;
      "23_WaitForSourceHeat" : SInt := 23;
      "24_PauseTime" : SInt := 24;
      "25_PowerControlZeroperformanceDemand" : SInt := 25;
      "26_HeatSink_Limit" : SInt := 26;
      "27_HeatSource_Limit" : SInt := 27;
      "28_VariableControl_Limit" : SInt := 28;
      "29_WaitingForShaftSeal" : SInt := 29;
      "210_State2DwellTime" : Int := 210;
      "30_PerformanceControlNotReady" : SInt := 30;
      "31_LubricationPrimingNotReady" : SInt := 31;
      "39_State3DwellTime" : SInt := 39;
      "50_WaitForOilHeat" : SInt := 50;
      "51_RampingUp" : SInt := 51;
      "52_DryingSuctionLine" : SInt := 52;
      "53_WaitForSuperHeatOut" : SInt := 53;
      "54_WaitForRecuperator" : SInt := 54;
      "55_SuctionManifoldPurge" : SInt := 55;
      "56_StartingAndHydrolock" : SInt := 56;
      "59_State4DwellTime" : SInt := 59;
      "60_Running" : SInt := 60;
      "61_State5DwellTime" : SInt := 61;
      "62_RunningAndHydrolock" : SInt := 62;
      "70_Stopping" : SInt := 70;
      "71_State7DwellTime" : SInt := 71;
      "72_StoppingDrySuctionLine" : SInt := 72;
      "302_PausedInState2" : Int := 302;
      "303_PausedInState3" : Int := 303;
      "304_PausedInState4" : Int := 304;
      "305_PausedInState5" : Int := 305;
      "307_PausedInState7" : Int := 307;
   END_VAR
   VAR_TEMP   // added for the SCL form of the ladder/FBD networks
      _w1 : Bool;
      _w2 : Bool;
   END_VAR
BEGIN

REGION Network 1 (SCL): Comments
   (* 
   What's with the fbWinCCTime & Time_Of_Day variables?

   When WinCC displays a TIME variable, it shows it as an integer number of milliseconds. So 5 minutes is 300,000ms. Not very intutive. 
   For longer times, like 1h20min, it's 4,800,000ms. To get a nice display of HH:MM:SS on the screen, and be able to enter time in this 
   format also, the Time_Of_Day variable type has to be used.

   All regulators & other structs use TIME because it's the right type to use, and the same is used everywhere for uniformity. WinCC 
   requires Time_Of_Day for usability. So instead of wrecking the structure and regularity of all those beautiful structs, a conversion 
   is done here (from TIME to TOD and back) to make TIME values "just work" in WinCC. It's ugly but it works, and frees the structs to be
   made the way the design requires, not the way WinCC requires.
   *)
END_REGION

REGION Network 2: Heartbeat
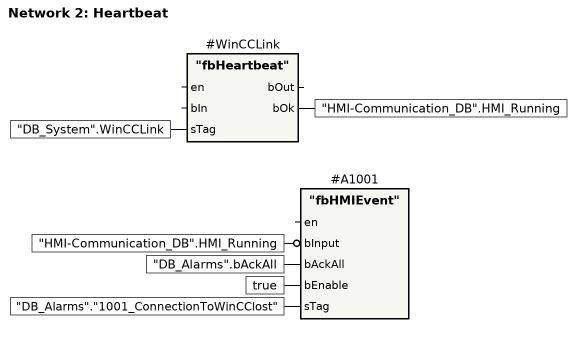
   #WinCCLink(sTag := "DB_System".WinCCLink, bOk => "HMI-Communication_DB".HMI_Running);   // "fbHeartbeat"
   #A1001(bInput := NOT "HMI-Communication_DB".HMI_Running,   // "fbHMIEvent"
          bAckAll := "DB_Alarms".bAckAll,
          bEnable := true,
          sTag := "DB_Alarms"."1001_ConnectionToWinCClost");
END_REGION

REGION Network 3: BackToStandby reason logic
   // Function to show, why the process fell back to standby
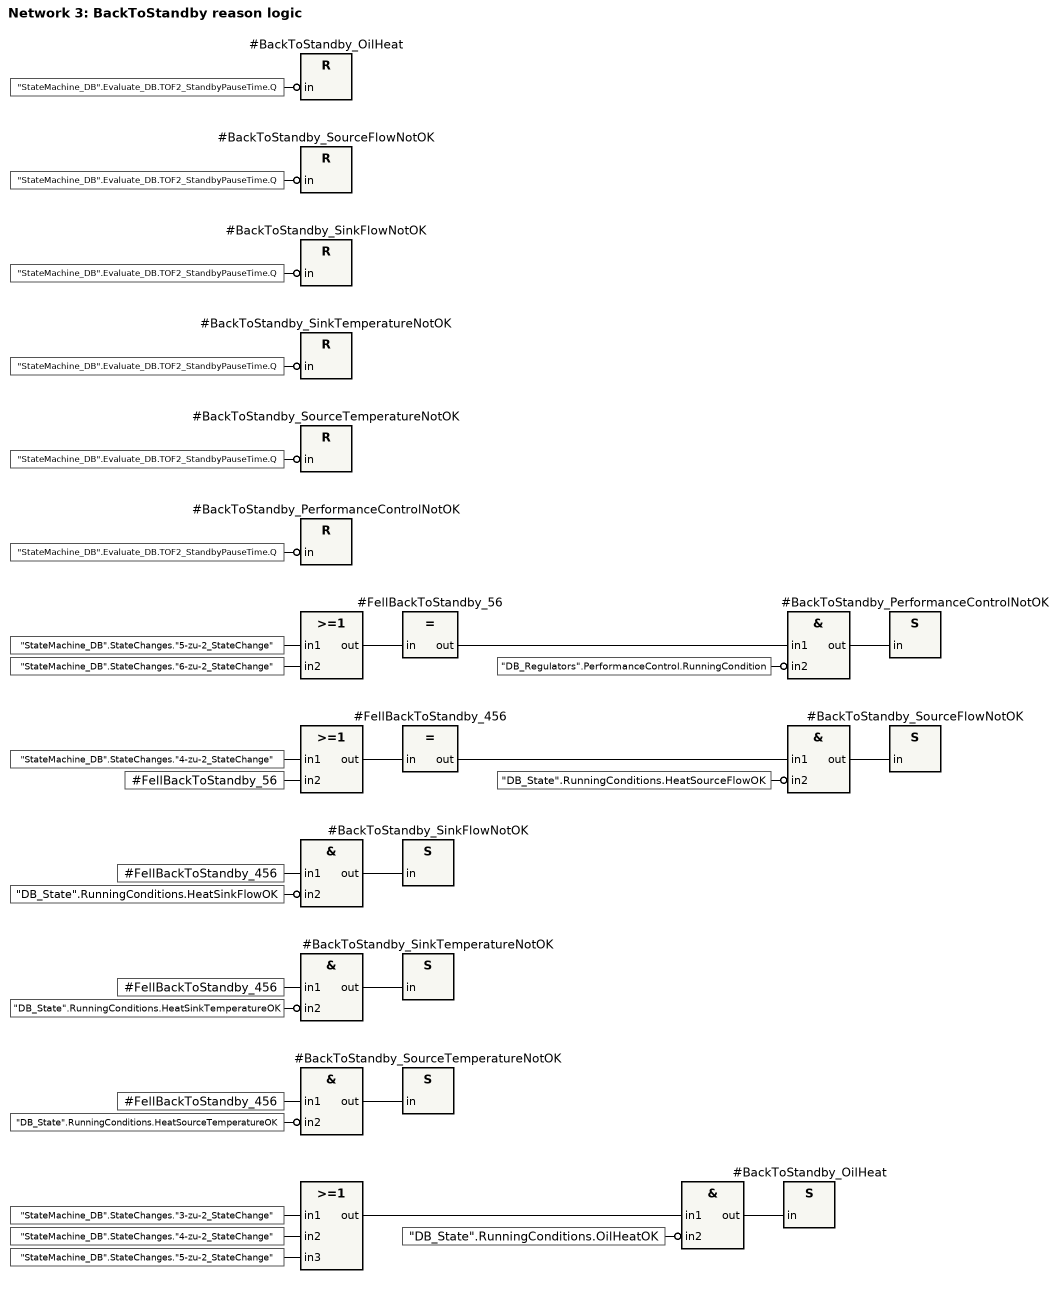
   IF NOT "StateMachine_DB".Evaluate_DB.TOF2_StandbyPauseTime.Q THEN
       #BackToStandby_OilHeat := FALSE;
       #BackToStandby_SourceFlowNotOK := FALSE;
       #BackToStandby_SinkFlowNotOK := FALSE;
       #BackToStandby_SinkTemperatureNotOK := FALSE;
       #BackToStandby_SourceTemperatureNotOK := FALSE;
       #BackToStandby_PerformanceControlNotOK := FALSE;
   END_IF;
   #FellBackToStandby_56 := "StateMachine_DB".StateChanges."5-zu-2_StateChange" OR "StateMachine_DB".StateChanges."6-zu-2_StateChange";
   IF #FellBackToStandby_56 AND NOT "DB_Regulators".PerformanceControl.RunningCondition THEN
       #BackToStandby_PerformanceControlNotOK := TRUE;
   END_IF;
   #FellBackToStandby_456 := "StateMachine_DB".StateChanges."4-zu-2_StateChange" OR #FellBackToStandby_56;
   IF #FellBackToStandby_456 AND NOT "DB_State".RunningConditions.HeatSourceFlowOK THEN
       #BackToStandby_SourceFlowNotOK := TRUE;
   END_IF;
   IF #FellBackToStandby_456 AND NOT "DB_State".RunningConditions.HeatSinkFlowOK THEN
       #BackToStandby_SinkFlowNotOK := TRUE;
   END_IF;
   IF #FellBackToStandby_456 AND NOT "DB_State".RunningConditions.HeatSinkTemperatureOK THEN
       #BackToStandby_SinkTemperatureNotOK := TRUE;
   END_IF;
   IF #FellBackToStandby_456 AND NOT "DB_State".RunningConditions.HeatSourceTemperatureOK THEN
       #BackToStandby_SourceTemperatureNotOK := TRUE;
   END_IF;
   IF ("StateMachine_DB".StateChanges."3-zu-2_StateChange" OR "StateMachine_DB".StateChanges."4-zu-2_StateChange" OR "StateMachine_DB".StateChanges."5-zu-2_StateChange") AND NOT "DB_State".RunningConditions.OilHeatOK THEN
       #BackToStandby_OilHeat := TRUE;
   END_IF;
END_REGION

REGION Network 4: BackToStandby-bit to trigger HMI-Message
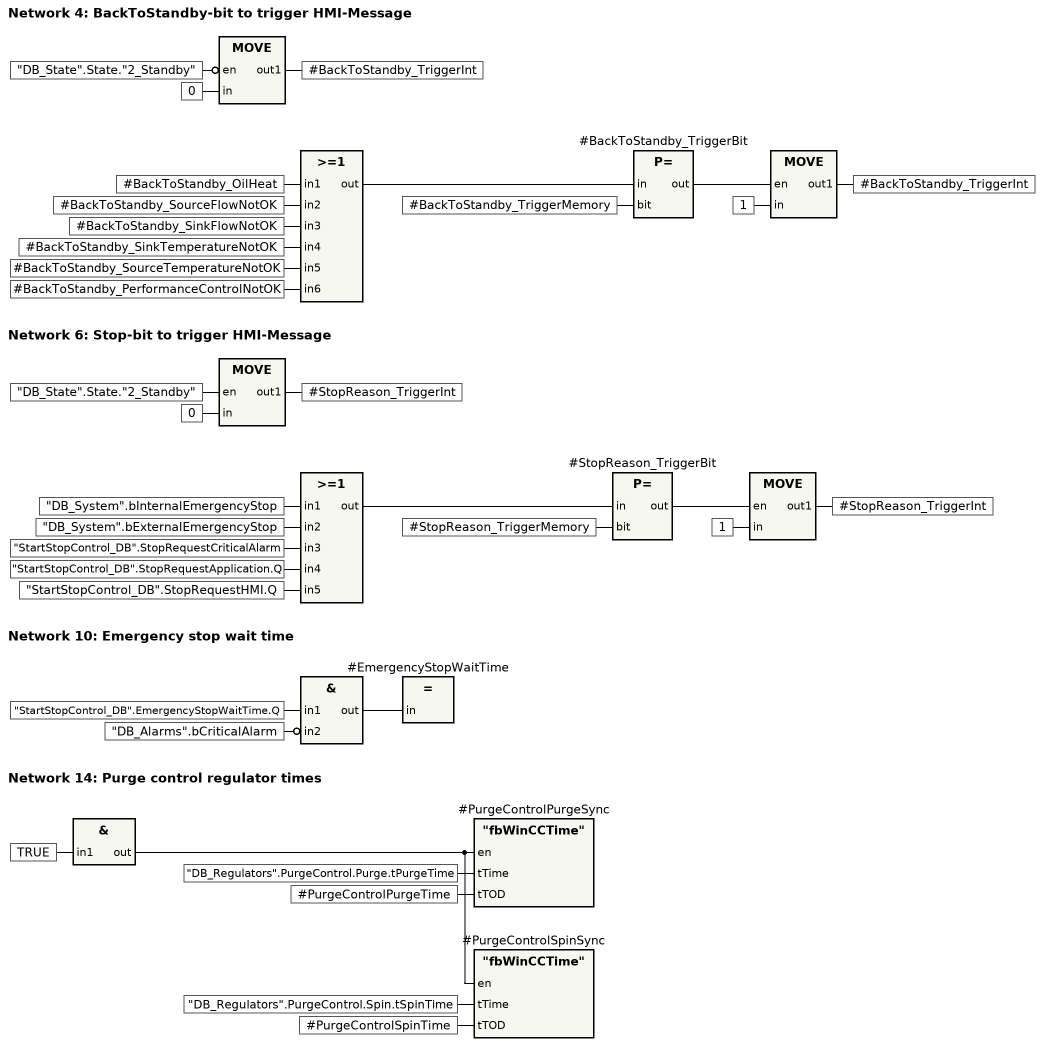
   IF NOT "DB_State".State."2_Standby" THEN #BackToStandby_TriggerInt := 0; END_IF;
   #_w1 := #BackToStandby_OilHeat OR #BackToStandby_SourceFlowNotOK OR #BackToStandby_SinkFlowNotOK OR #BackToStandby_SinkTemperatureNotOK OR #BackToStandby_SourceTemperatureNotOK OR #BackToStandby_PerformanceControlNotOK;
   #BackToStandby_TriggerBit := #_w1 AND NOT #BackToStandby_TriggerMemory;   // rising edge
   #BackToStandby_TriggerMemory := #_w1;
   IF #_w1 THEN #BackToStandby_TriggerInt := 1; END_IF;
END_REGION

REGION Network 5 (SCL): BackToStandby reason text
   // Write "back-to-standby" reason to text and deliver it to the HMI
   IF #BackToStandby_OilHeat THEN
       #BackToStandbyReason_Text := 'Oil heat was not OK!';
   ELSIF #BackToStandby_PerformanceControlNotOK THEN
       #BackToStandbyReason_Text := 'No power was required!';
   ELSIF #BackToStandby_SourceTemperatureNotOK THEN
       #BackToStandbyReason_Text := 'Heat source was not OK!';
   ELSIF #BackToStandby_SinkTemperatureNotOK THEN
       #BackToStandbyReason_Text := 'Heat sink was not OK!';
   ELSIF #BackToStandby_SourceFlowNotOK THEN
       #BackToStandbyReason_Text := 'No source mass flow!';
   ELSIF #BackToStandby_SinkFlowNotOK THEN
       #BackToStandbyReason_Text := 'No sink mass flow!';
   ELSE
       #BackToStandbyReason_Text := '';
   END_IF;
END_REGION

REGION Network 6: Stop-bit to trigger HMI-Message
   IF "DB_State".State."2_Standby" THEN #StopReason_TriggerInt := 0; END_IF;
   #_w1 := "DB_System".bInternalEmergencyStop OR "DB_System".bExternalEmergencyStop OR "StartStopControl_DB".StopRequestCriticalAlarm OR "StartStopControl_DB".StopRequestApplication.Q OR "StartStopControl_DB".StopRequestHMI.Q;
   #StopReason_TriggerBit := #_w1 AND NOT #StopReason_TriggerMemory;   // rising edge
   #StopReason_TriggerMemory := #_w1;
   IF #_w1 THEN #StopReason_TriggerInt := 1; END_IF;
END_REGION

REGION Network 7 (SCL): Stop reason text
   // Write stop reason to text and deliver it to the HMI
   IF "DB_System".bInternalEmergencyStop THEN
       //Emergency Stop intern
       #StopReason_Text := 'Internal emergency stopp!';
   ELSIF "DB_System".bExternalEmergencyStop THEN
       //Emergency Stop extern
       #StopReason_Text := 'External emergency stopp!';
   ELSIF "StartStopControl_DB".StopRequestCriticalAlarm THEN
       //Stop via critical alarm 
       #StopReason_Text := 'Critical alarm!';
   ELSIF "StartStopControl_DB".StopRequestApplication.Q THEN
       //Stop via application PLC
       #StopReason_Text := 'External stopp request!';
   ELSIF "StartStopControl_DB".StopRequestHMI.Q THEN
       //Stop via HMI  
       #StopReason_Text := 'HMI stopp request!';
   END_IF;
END_REGION

REGION Network 8 (SCL): State text & progress text
   // #Progress_Text = 1 is the catch-all error state. If you end up there then there is more work to do.
   CASE "DB_State".State.State_Number OF
       0:  #State_Text := 'Init';

           IF "DB_State".SystemInitialised = FALSE THEN
               #Progress_Text := #"05_CPU_Init";
           ELSE
               #Progress_Text := #"01_WaitingForStateChange";
           END_IF;

       1:  #State_Text := 'Offline';

           IF "DB_System".bEmergencyStop = TRUE THEN
               #Progress_Text := #"11_EmergencyStopActive";
           ELSIF "DB_Alarms"."1110_HBL_SC_10_CommError".sState.bActive OR "DB_Alarms"."1130_HBL_SC_10_Tripped".sState.bActive THEN
               #Progress_Text := #"12_InverterNotOnline";
           ELSIF "DB_Alarms".bCriticalAlarm = TRUE THEN
               #Progress_Text := #"6_CriticalAlarmActive";
           ELSIF "StartStopControl_DB".EmergencyStopWaitTime.Q = TRUE THEN
               #Progress_Text := #"14_EmergencyStopWaitTime";
           ELSIF "DB_Alarms".bCommonAlarm = TRUE THEN
               #Progress_Text := #"13_ReadyToStartWithActiveWarnings";
           ELSE
               #Progress_Text := #"10_ReadyToStart";
           END_IF;


       2:  #State_Text := 'Standby';

           IF "DB_State".RunningConditions.HeatSourceFlowOK = FALSE THEN
               #Progress_Text := #"20_WaitForSourceFlow";
           ELSIF "DB_State".RunningConditions.HeatSinkFlowOK = FALSE THEN
               #Progress_Text := #"21_WaitForSinkFlow";
           ELSIF "DB_State".RunningConditions.HeatSinkTemperatureOK = FALSE THEN
               #Progress_Text := #"22_WaitForSinkHeat";
           ELSIF "DB_State".RunningConditions.HeatSourceTemperatureOK = FALSE THEN
               #Progress_Text := #"23_WaitForSourceHeat";
           ELSIF "StateMachine_DB".Evaluate_DB.TOF2_StandbyPauseTime.Q = TRUE THEN
               #Progress_Text := #"24_PauseTime";
           ELSIF "StateMachine_DB".Evaluate_DB.TON2_Standby.Q = FALSE THEN
               #Progress_Text :=#"210_State2DwellTime";
           ELSIF "DB_Regulators".PerformanceControl.RunningCondition = FALSE THEN
               IF "Regulation_DB".PerformanceControl.HeatSinkTimer.Q = FALSE THEN
                   #Progress_Text := #"26_HeatSink_Limit";
               ELSIF ("Regulation_DB".PerformanceControl.HeatSourceTimer.Q) = FALSE THEN
                   #Progress_Text := #"27_HeatSource_Limit";
               ELSIF "Regulation_DB".PerformanceControl.VariableControlTimer.Q = FALSE THEN
                   #Progress_Text := #"28_VariableControl_Limit";
               ELSE
                   #Progress_Text := #"25_PowerControlZeroperformanceDemand";
               END_IF;
           ELSIF "DB_State".StatePauseFlags[2] = TRUE THEN
               #Progress_Text := #"302_PausedInState2";
           ELSE
               #Progress_Text := #"01_WaitingForStateChange";
           END_IF;

       3:  #State_Text := 'Prepare Start';

           IF "DB_State".RunningConditions.ShaftSealSystemOK = FALSE THEN
               #Progress_Text := #"29_WaitingForShaftSeal";
           ELSIF "DB_State".RunningConditions.OilHeatOK = FALSE THEN
               #Progress_Text := #"50_WaitForOilHeat";
           ELSIF "DB_State".RunningConditions.LubricationPrimingOk = FALSE THEN
               #Progress_Text := #"31_LubricationPrimingNotReady";
           ELSIF "DB_Regulators".PerformanceControl.RunningCondition = FALSE THEN
               #Progress_Text := #"30_PerformanceControlNotReady";
           ELSIF "StateMachine_DB".Evaluate_DB.TON3_PrepareStart.Q = FALSE THEN
               #Progress_Text := #"39_State3DwellTime";
           ELSIF "DB_State".StatePauseFlags[3] = TRUE THEN
               #Progress_Text := #"303_PausedInState3";
           ELSE
               #Progress_Text := #"01_WaitingForStateChange";
           END_IF;

       4:  #State_Text := 'Starting';

           IF "DB_State".RunningConditions.DoWarmStart = FALSE AND "DB_Regulators".PurgeControl.bDone = FALSE THEN
               #Progress_Text := #"55_SuctionManifoldPurge";
           ELSIF "DB_State".RunningConditions.AtOrAboveHydrolockSpeed = FALSE THEN
               #Progress_Text := #"51_RampingUp";
           ELSIF "DB_State".RunningConditions.SuctionLineDry = FALSE THEN
               #Progress_Text := #"52_DryingSuctionLine";
           ELSIF "StateMachine_DB".Evaluate_DB.TON4_Start.Q = FALSE THEN
               #Progress_Text := #"59_State4DwellTime";
           ELSIF "DB_State".StatePauseFlags[4] = TRUE THEN
               #Progress_Text := #"304_PausedInState4";
           ELSE
               #Progress_Text := #"01_WaitingForStateChange";
           END_IF;

       5:  #State_Text := 'Warm-up';

           IF "DB_State".RunningConditions.RiskOfHydrolock = TRUE THEN
               #Progress_Text := #"56_StartingAndHydrolock";
           ELSIF "DB_State".RunningConditions.SuperheatCompressorOutOK = FALSE THEN
               #Progress_Text := #"53_WaitForSuperHeatOut";
           ELSIF "DB_State".RunningConditions.RecuperatorWorking = FALSE THEN
               #Progress_Text := #"54_WaitForRecuperator";
           ELSIF "StateMachine_DB".Evaluate_DB.TON5_Warmup.Q = FALSE THEN
               #Progress_Text := #"61_State5DwellTime";
           ELSIF "DB_State".StatePauseFlags[5] = TRUE THEN
               #Progress_Text := #"305_PausedInState5";
           ELSE
               #Progress_Text := #"01_WaitingForStateChange";
           END_IF;

       6:  #State_Text := 'Running';
           IF "DB_State".RunningConditions.RiskOfHydrolock = TRUE THEN
               #Progress_Text := #"62_RunningAndHydrolock";
           ELSE
               #Progress_Text := #"60_Running";
           END_IF;

       7:  #State_Text := 'Stop';

           IF "DB_State".RunningConditions.SuctionLineDry = FALSE AND"DB_State".FastStop = FALSE THEN
               #Progress_Text := #"72_StoppingDrySuctionLine";
           ELSIF "DB_InverterDrives".HBL_SC_10.Stat.Speed.Eng.fValue <> 0 THEN
               #Progress_Text := #"70_Stopping";
           ELSIF "StateMachine_DB".Evaluate_DB.TON7_Stop.Q = FALSE THEN
               #Progress_Text := #"71_State7DwellTime";
           ELSE
               #Progress_Text := #"01_WaitingForStateChange";
           END_IF;

       ELSE  
           #State_Text := 'No state!';
   END_CASE;
END_REGION

REGION Network 9 (SCL): Regulation target
   // Repeating some of the logic from PerformanceControl (FB9) here, making it fragile
   // Conditions are evaluated as repeated IFs and not ELSIFs because that is how it is evaluated in FB9. Yes, confusing.
   // This network provides an alternative interface to Performance Control, using its public API (DB_Regulators.PerformanceControl)
   // Figure out which target is active & select setpoint
   IF "DB_Regulators".PerformanceControl.Settings.HeatSink.Control_Active THEN
       IF "DB_Regulators".PerformanceControl.Settings.HeatSink.UseFeedFlow THEN
           #RegulationTarget := 2;
       ELSE
           #RegulationTarget := 1;
       END_IF;
   END_IF;

   IF "DB_Regulators".PerformanceControl.Settings.HeatSource.Control_Active THEN
       IF "DB_Regulators".PerformanceControl.Settings.HeatSource.UseFeedFlow THEN
           #RegulationTarget := 4;
       ELSE
           #RegulationTarget := 3;
       END_IF;
   END_IF;

   IF "DB_Regulators".PerformanceControl.Settings.VariableControl.Control_Active AND "DB_Regulators".PerformanceControl.Settings.VariableControl.ReferenceID > 0 THEN
       #RegulationTarget := 6;
   END_IF;

   // Update the currently selected setpoint if updated from HMI
   IF #HeatboosterSetpoint <> #HeatboosterSetpointPrev THEN
       // Select the right setpoint
       CASE #RegulationTarget OF
       1..2 : "DB_Regulators".PerformanceControl.Settings.HeatSink.Setpoint := #HeatboosterSetpoint;
       3..4 : "DB_Regulators".PerformanceControl.Settings.HeatSource.Setpoint := #HeatboosterSetpoint;
       6    : "DB_Regulators".PerformanceControl.Settings.VariableControl.Setpoint := #HeatboosterSetpoint;
       END_CASE;
   END_IF;
   #HeatboosterSetpointPrev := #HeatboosterSetpoint;
END_REGION

REGION Network 10: Emergency stop wait time
   // Do not show when a critical alarm is active
   #EmergencyStopWaitTime := "StartStopControl_DB".EmergencyStopWaitTime.Q AND NOT "DB_Alarms".bCriticalAlarm;
END_REGION

REGION Network 11 (SCL): Emergency lock time
   // Gruesome, this needs refactoring
   #EmergencyStopCountdown := TIME_TO_TOD(IN := ("StartStopControl_DB".EmergencyStopWaitTime.PT - "StartStopControl_DB".EmergencyStopWaitTime.ET));
   IF #SkipEmergencyStopWait THEN
       RESET_TIMER("StartStopControl_DB".EmergencyStopWaitTime);
   END_IF;
END_REGION

REGION Network 12 (SCL): Dwell times
   #State2DwellTimeElapsed := TIME_TO_TOD("StateMachine_DB".Evaluate_DB.TON2_Standby.ET);
   #State2DwellSync(tTime := "DB_CurrentSetting".MissingSetting.Misc.State2DwellTime, tTOD := #State2DwellTime);

   #State3DwellTimeElapsed := TIME_TO_TOD("StateMachine_DB".Evaluate_DB.TON3_PrepareStart.ET);
   #State3DwellSync(tTime := "DB_CurrentSetting".MissingSetting.Misc.State3DwellTime, tTOD := #State3DwellTime);

   #State4DwellTimeElapsed := TIME_TO_TOD("StateMachine_DB".Evaluate_DB.TON4_Start.ET);
   #State4DwellSync(tTime := "DB_CurrentSetting".MissingSetting.Misc.State4DwellTime, tTOD := #State4DwellTime);

   #State5DwellTimeElapsed := TIME_TO_TOD("StateMachine_DB".Evaluate_DB.TON5_Warmup.ET);
   #State5DwellSync(tTime := "DB_CurrentSetting".MissingSetting.Misc.State5DwellTime, tTOD := #State5DwellTime);

   #State7DwellTimeElapsed := TIME_TO_TOD("StateMachine_DB".Evaluate_DB.TON7_Stop.ET);
   #State7DwellSync(tTime := "DB_CurrentSetting".MissingSetting.Misc.State7DwellTime, tTOD := #State7DwellTime);
END_REGION

REGION Network 13 (SCL): Pause time
   #State2PauseTimeElapsed := TIME_TO_TOD("StateMachine_DB".Evaluate_DB.TOF2_StandbyPauseTime.ET);
   #State2PauseSync(tTime := "DB_CurrentSetting".MissingSetting.Misc.State2PauseTime, tTOD := #State2PauseTime);
END_REGION

REGION Network 14: Purge control regulator times
   IF TRUE THEN
       #PurgeControlPurgeSync(tTime := "DB_Regulators".PurgeControl.Purge.tPurgeTime,   // "fbWinCCTime"
                              tTOD := #PurgeControlPurgeTime);
       #PurgeControlSpinSync(tTime := "DB_Regulators".PurgeControl.Spin.tSpinTime, tTOD := #PurgeControlSpinTime);   // "fbWinCCTime"
   END_IF;
END_REGION

REGION Network 15: CPC progressive regulator
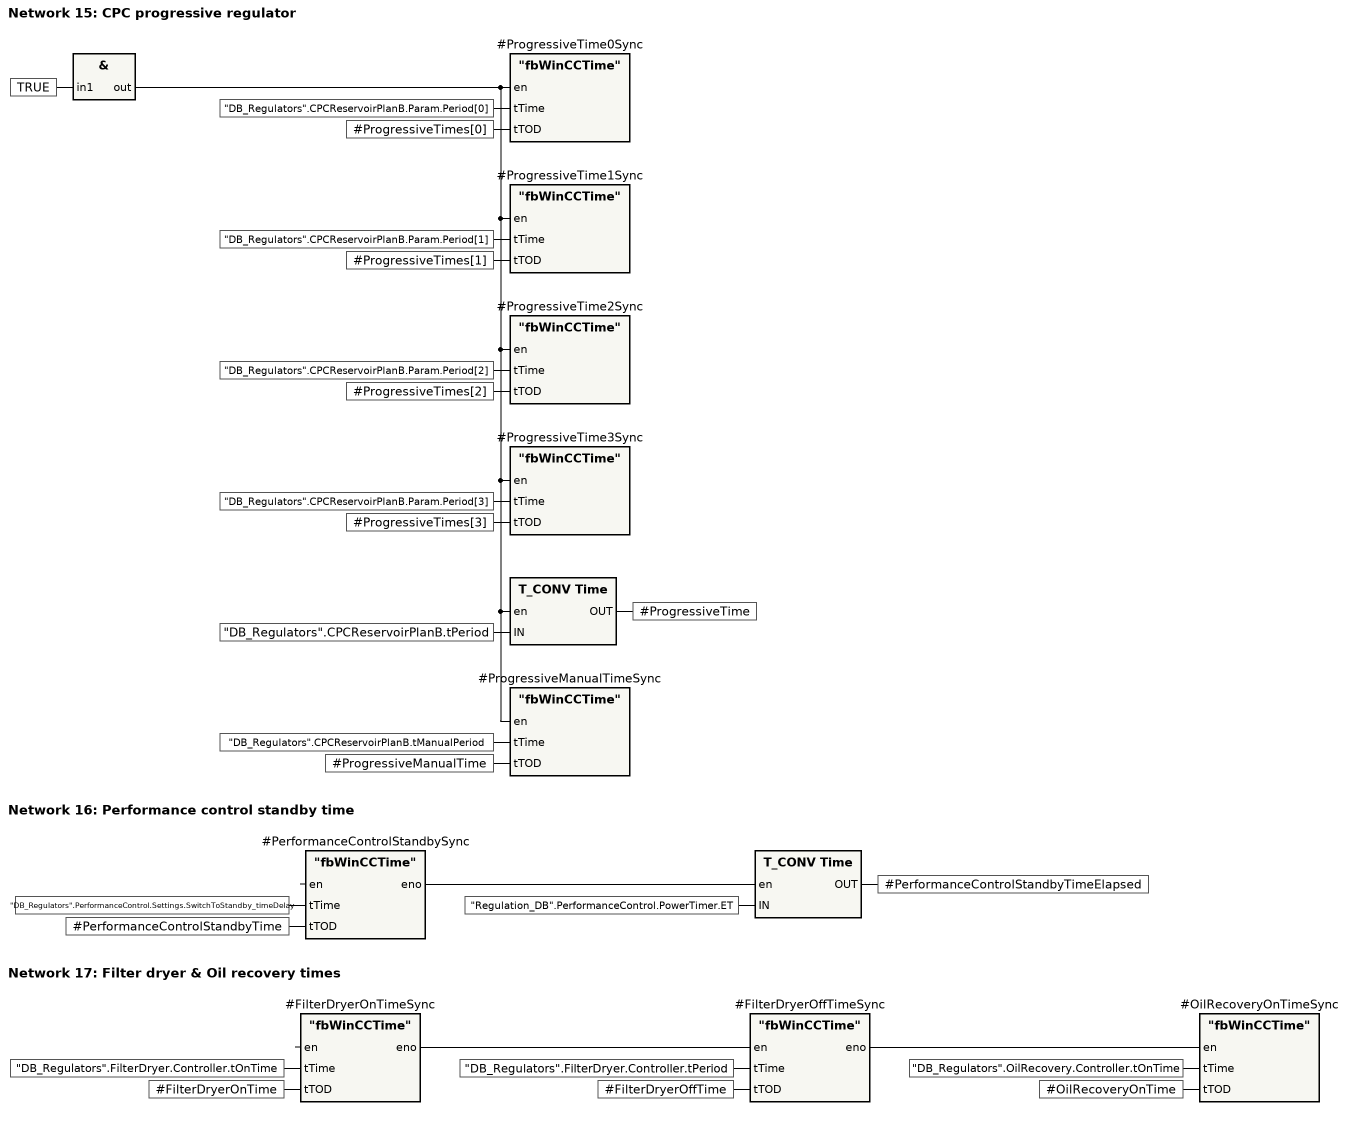
   IF TRUE THEN
       #ProgressiveTime0Sync(tTime := "DB_Regulators".CPCReservoirPlanB.Param.Period[0],   // "fbWinCCTime"
                             tTOD := #ProgressiveTimes[0]);
       #ProgressiveTime1Sync(tTime := "DB_Regulators".CPCReservoirPlanB.Param.Period[1],   // "fbWinCCTime"
                             tTOD := #ProgressiveTimes[1]);
       #ProgressiveTime2Sync(tTime := "DB_Regulators".CPCReservoirPlanB.Param.Period[2],   // "fbWinCCTime"
                             tTOD := #ProgressiveTimes[2]);
       #ProgressiveTime3Sync(tTime := "DB_Regulators".CPCReservoirPlanB.Param.Period[3],   // "fbWinCCTime"
                             tTOD := #ProgressiveTimes[3]);
       T_CONV(IN := "DB_Regulators".CPCReservoirPlanB.tPeriod, OUT => #ProgressiveTime);
       #ProgressiveManualTimeSync(tTime := "DB_Regulators".CPCReservoirPlanB.tManualPeriod,   // "fbWinCCTime"
                               tTOD := #ProgressiveManualTime);
   END_IF;
END_REGION

REGION Network 16: Performance control standby time
   #PerformanceControlStandbySync(tTime := "DB_Regulators".PerformanceControl.Settings.SwitchToStandby_timeDelay,   // "fbWinCCTime"
                           tTOD := #PerformanceControlStandbyTime,
                           ENO => #_w1);
   IF #_w1 THEN
       T_CONV(IN := "Regulation_DB".PerformanceControl.PowerTimer.ET, OUT => #PerformanceControlStandbyTimeElapsed);
   END_IF;
END_REGION

REGION Network 17: Filter dryer & Oil recovery times
   #FilterDryerOnTimeSync(tTime := "DB_Regulators".FilterDryer.Controller.tOnTime,   // "fbWinCCTime"
                          tTOD := #FilterDryerOnTime,
                          ENO => #_w1);
   #FilterDryerOffTimeSync(EN := #_w1,   // "fbWinCCTime"
                           tTime := "DB_Regulators".FilterDryer.Controller.tPeriod,
                           tTOD := #FilterDryerOffTime,
                           ENO => #_w2);
   IF #_w2 THEN
       #OilRecoveryOnTimeSync(tTime := "DB_Regulators".OilRecovery.Controller.tOnTime, tTOD := #OilRecoveryOnTime);   // "fbWinCCTime"
   END_IF;
END_REGION

REGION Network 18: Process Valves
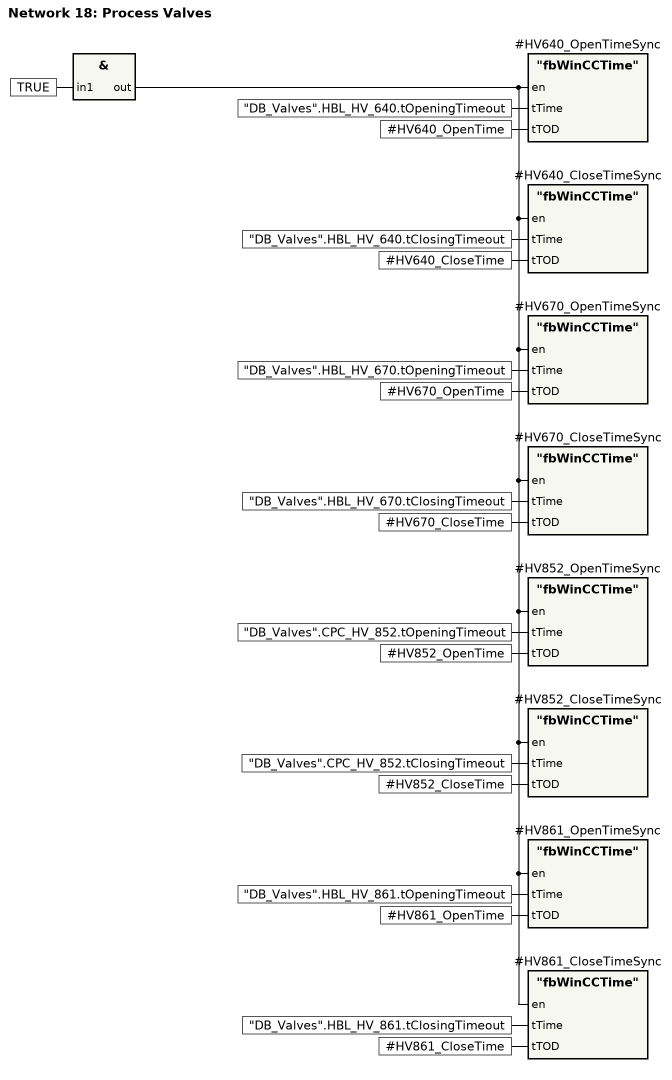
   IF TRUE THEN
       #HV640_OpenTimeSync(tTime := "DB_Valves".HBL_HV_640.tOpeningTimeout, tTOD := #HV640_OpenTime);   // "fbWinCCTime"
       #HV640_CloseTimeSync(tTime := "DB_Valves".HBL_HV_640.tClosingTimeout, tTOD := #HV640_CloseTime);   // "fbWinCCTime"
       #HV670_OpenTimeSync(tTime := "DB_Valves".HBL_HV_670.tOpeningTimeout, tTOD := #HV670_OpenTime);   // "fbWinCCTime"
       #HV670_CloseTimeSync(tTime := "DB_Valves".HBL_HV_670.tClosingTimeout, tTOD := #HV670_CloseTime);   // "fbWinCCTime"
       #HV852_OpenTimeSync(tTime := "DB_Valves".CPC_HV_852.tOpeningTimeout, tTOD := #HV852_OpenTime);   // "fbWinCCTime"
       #HV852_CloseTimeSync(tTime := "DB_Valves".CPC_HV_852.tClosingTimeout, tTOD := #HV852_CloseTime);   // "fbWinCCTime"
       #HV861_OpenTimeSync(tTime := "DB_Valves".HBL_HV_861.tOpeningTimeout, tTOD := #HV861_OpenTime);   // "fbWinCCTime"
       #HV861_CloseTimeSync(tTime := "DB_Valves".HBL_HV_861.tClosingTimeout, tTOD := #HV861_CloseTime);   // "fbWinCCTime"
   END_IF;
END_REGION
END_FUNCTION_BLOCK

FUNCTION_BLOCK "fbHeartbeat"
{ S7_Optimized_Access := 'TRUE' }
VERSION : 0.1
   VAR_INPUT 
      bIn : Bool;   // Signal from partner
   END_VAR

   VAR_OUTPUT 
      bOut : Bool;   // Signal to partner
      bOk : Bool;
   END_VAR

   VAR_IN_OUT 
      sTag : "stHeartbeat";
   END_VAR

   VAR 
      Timeout {InstructionName := 'TON_TIME'; LibVersion := '1.0'; S7_SetPoint := 'False'} : TON_TIME;
   END_VAR

   VAR_TEMP 
      In : Bool;
   END_VAR


BEGIN
	// fbHeartbeat - communications monitoring
	// Send a bit back and forth. This side does all the work, the other side just sends back what it has gotten.
	// bOut is set, and waits for bIn to be set before the timeout.
	// Then bOut is cleared and waits for bIn to be cleared before the timeout. 
	
	// Combine local & tag input sources
	#In := #bIn OR #sTag.bIn;
	
	// Timeout
	#Timeout(IN := (#sTag.nState = 2), PT := #sTag.tTimeout);
	
	// States
	CASE #sTag.nState OF
	    0: // Idle
	        #sTag.bOut := FALSE;
	        IF #sTag.bEnable = TRUE THEN
	            #sTag.nState := 1;
	        END_IF;
	    1: // Ping
	        #sTag.bOut := #sTag.bOut XOR TRUE;
	        IF #sTag.bEnable = FALSE THEN
	            #sTag.nState := 0;
	        ELSE
	            #sTag.nState := 2;
	            #sTag.bOk := TRUE;
	        END_IF;
	    2: // Wait
	        IF #In = #sTag.bOut THEN
	            // Pong
	            #sTag.nState := 1;
	        ELSIF #Timeout.Q = TRUE THEN
	            #sTag.nState := 3;
	            #sTag.bOk := FALSE;
	        ELSIF #sTag.bEnable = FALSE THEN
	            #sTag.nState := 0;
	        END_IF;
	    3: // Timeout
	        IF #In = #sTag.bOut THEN
	            #sTag.nState := 1;
	            #sTag.bOk := TRUE;
	        ELSIF #sTag.bEnable = FALSE THEN
	            #sTag.nState := 0;
	        END_IF;
	        
	END_CASE;
	
	// Local outputs
	#bOut := #sTag.bOut;
	#bOk := #sTag.bOk;
	
	
	
END_FUNCTION_BLOCK

FUNCTION_BLOCK "fbWinCCTime"
{ S7_Optimized_Access := 'TRUE' }
AUTHOR : Heaten
VERSION : 0.1
   VAR_IN_OUT 
      tTime : Time;   // The source time value
      tTOD : Time_Of_Day;   // The TOD value in the HMI
   END_VAR

   VAR 
      tTime_prev : Time;
      tTOD_prev : Time_Of_Day;
   END_VAR


BEGIN
	// Allow displaying & modifying of a TIME value in WinCC
	// TIME is displayed as an integer representing milliseconds, which is usually not what you want
	// TOD is represented hh:mm:ss and can also be entered in this format, which is usually what you want
	
	IF #tTOD <> #tTOD_prev THEN
	    // updated from HMI, update the PLC value
	    #tTime := TOD_TO_TIME(#tTOD);
	ELSIF #tTime <> #tTime_prev THEN
	    // updated from the PLC, update the HMI value
	    #tTOD := TIME_TO_TOD(#tTime);
	END_IF;
	
	// update
	#tTOD_prev := #tTOD;
	#tTime_prev := #tTime;
END_FUNCTION_BLOCK

FUNCTION "SoftwareVersion" : String
{ S7_Optimized_Access := 'TRUE' }
AUTHOR : Heaten
VERSION : 0.1

BEGIN
	// SOFTWARE VERSION: in-band software change tracking
	// Changes and descriptions are usually tracked out-of-band, eg as git commit messages or as issues in github etc. This is to more tightly couple change tracking with the actual project.
	// INSTRUCTIONS:
	// 1. New entries should go at the top, such that the most recent changes are visible first.
	// 2. Be short but descriptive; one line per change is a good starting point.
	// 3. Change the version number. This is a string so there is a lot of flexibility as to the format.
	
	#SoftwareVersion := 'V5.0.1.1';
	
	//V5.0.1.1
	//16.05.2025 Birk
	//Wrong value in FB9 PerformanceControl Network 7 Line 5 fixed
	//Changes in Application PLC
	
	// V5.0.1.0
	// 12.05.2025 12:00 Birk
	// Task #7 Last stop reason
	// Added memory space for triggers and text in DB3 HMI-Communication_DB
	// Added networks with code in FB3 HMI-Communication to trigger a Stop and write its reason to a text
	// Added events in HMI including variables from PLC and activated Events in Alarm screens
	// 07.05.2025 12:00 Birk
	// Task #4 "POWER CONTROL - Gain factor"
	// Removed abs() from FB9 Performance Control: Heat Sink, Heat Source, Variable controller
	// Instead of setting controller gain to 1.0, recalculation of ControllerError before actual controller
	// Adjustment of Kp in DB18 DB_Regulators.PerformanceControl.Settings and FB5_Regulation like specified in Git task
	// Added Watch table Simulation_Offenau_OFF
	// 08.05.2025 12:00 Birk
	// Task #6 "Visualisize Power control"
	// Added text field to HMI Screen "Performance Control" which shows a text depending on current power limitation
	// Added watch table "BypassApplCom"
	// Fixed wrong scaling factors in DB_AI for a few "TT"
	
	// V5.0.0.0 28.03.2025
	// - forked from Alpha-2 V4.0.0.7
	// - V5 is for the split-system steam/steam
	// - updated hardware to include RIO1, RIO2, subset of "Sensors" which is now just the shaft seal system
	// - updated sensor claibration ranges where known
	// - added processing in & out for all new instruments
	
	
END_FUNCTION

ORGANIZATION_BLOCK "Main_Cyclic"   // OB35, FBD, CyclicInterrupt
TITLE = Realtime task
{ S7_Optimized_Access := 'TRUE' }
VERSION : 0.1
// stored: AutoNumber false, IsIECCheckEnabled false, SetENOAutomatically false
   VAR_INPUT
      Initial_Call : Bool;
      Event_Count : Int;
   END_VAR
BEGIN

REGION Network 1
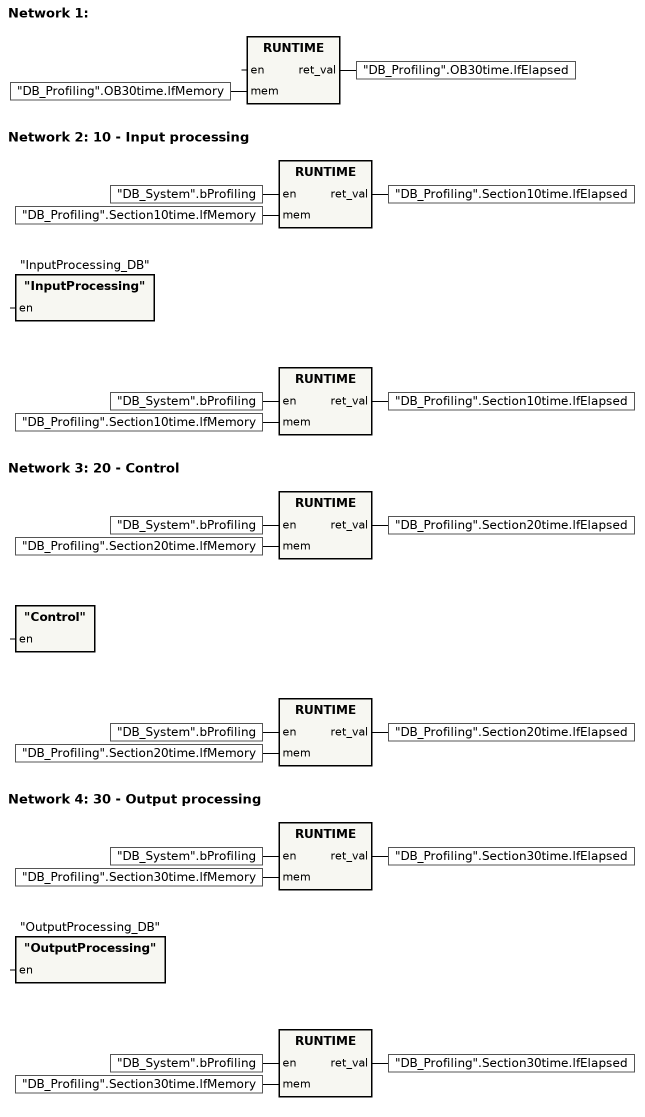
   // no SCL statement known for Runtime: written as a call
   "DB_Profiling".OB30time.lfElapsed := Runtime(mem := "DB_Profiling".OB30time.lfMemory);
END_REGION

REGION Network 2: 10 - Input processing
   // no SCL statement known for Runtime: written as a call
   IF "DB_System".bProfiling THEN
       "DB_Profiling".Section10time.lfElapsed := Runtime(mem := "DB_Profiling".Section10time.lfMemory);
   END_IF;
   "InputProcessing_DB"();   // "InputProcessing"
   IF "DB_System".bProfiling THEN
       "DB_Profiling".Section10time.lfElapsed := Runtime(mem := "DB_Profiling".Section10time.lfMemory);
   END_IF;
END_REGION

REGION Network 3: 20 - Control
   // no SCL statement known for Runtime: written as a call
   IF "DB_System".bProfiling THEN
       "DB_Profiling".Section20time.lfElapsed := Runtime(mem := "DB_Profiling".Section20time.lfMemory);
   END_IF;
   "Control"();
   IF "DB_System".bProfiling THEN
       "DB_Profiling".Section20time.lfElapsed := Runtime(mem := "DB_Profiling".Section20time.lfMemory);
   END_IF;
END_REGION

REGION Network 4: 30 - Output processing
   // no SCL statement known for Runtime: written as a call
   IF "DB_System".bProfiling THEN
       "DB_Profiling".Section30time.lfElapsed := Runtime(mem := "DB_Profiling".Section30time.lfMemory);
   END_IF;
   "OutputProcessing_DB"();   // "OutputProcessing"
   IF "DB_System".bProfiling THEN
       "DB_Profiling".Section30time.lfElapsed := Runtime(mem := "DB_Profiling".Section30time.lfMemory);
   END_IF;
END_REGION

REGION Network 5: 40 - Alarms
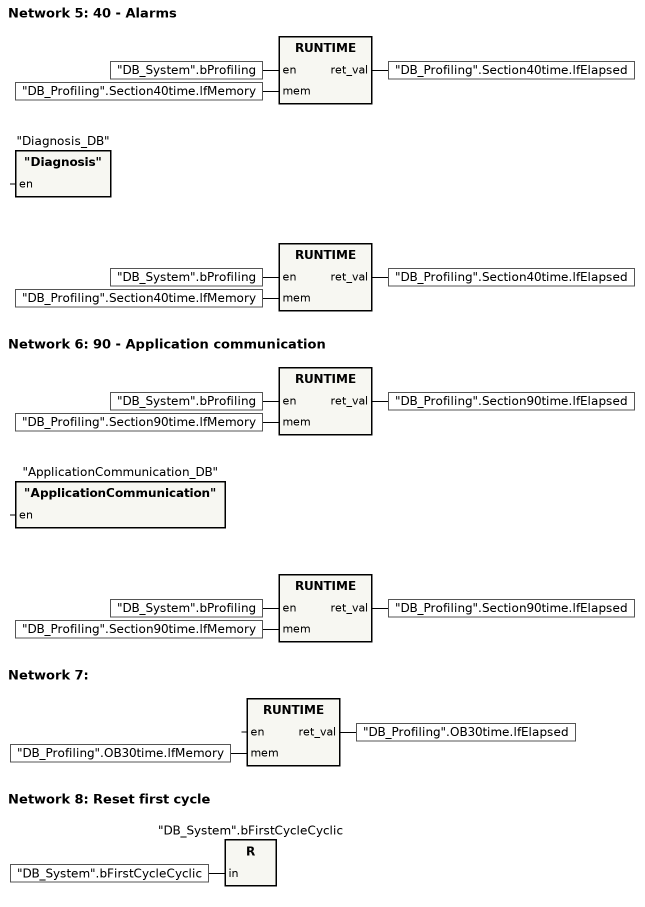
   // no SCL statement known for Runtime: written as a call
   IF "DB_System".bProfiling THEN
       "DB_Profiling".Section40time.lfElapsed := Runtime(mem := "DB_Profiling".Section40time.lfMemory);
   END_IF;
   "Diagnosis_DB"();   // "Diagnosis"
   IF "DB_System".bProfiling THEN
       "DB_Profiling".Section40time.lfElapsed := Runtime(mem := "DB_Profiling".Section40time.lfMemory);
   END_IF;
END_REGION

REGION Network 6: 90 - Application communication
   // Exchange data with the Application PLC
   // no SCL statement known for Runtime: written as a call
   IF "DB_System".bProfiling THEN
       "DB_Profiling".Section90time.lfElapsed := Runtime(mem := "DB_Profiling".Section90time.lfMemory);
   END_IF;
   "ApplicationCommunication_DB"();   // "ApplicationCommunication"
   IF "DB_System".bProfiling THEN
       "DB_Profiling".Section90time.lfElapsed := Runtime(mem := "DB_Profiling".Section90time.lfMemory);
   END_IF;
END_REGION

REGION Network 7
   // no SCL statement known for Runtime: written as a call
   "DB_Profiling".OB30time.lfElapsed := Runtime(mem := "DB_Profiling".OB30time.lfMemory);
END_REGION

REGION Network 8: Reset first cycle
   // This network must be the last one in the program
   IF "DB_System".bFirstCycleCyclic THEN "DB_System".bFirstCycleCyclic := FALSE; END_IF;
END_REGION
END_ORGANIZATION_BLOCK

FUNCTION_BLOCK "InputProcessing"   // FB48, FBD
{ S7_Optimized_Access := 'TRUE' }
AUTHOR : Heaten
VERSION : 0.1
// stored: AutoNumber true, IsIECCheckEnabled false, IsRetainMemResEnabled false, MemoryReserve 0, SetENOAutomatically false, UDAEnableTagReadback false
   VAR
      AnalogInputProcessing_DB { ExternalAccessible := 'False'; ExternalVisible := 'False'; ExternalWritable := 'False'} : "AnalogInputProcessing";
      InputAlarmHandling_DB { ExternalAccessible := 'False'; ExternalVisible := 'False'; ExternalWritable := 'False'} : "InputAlarmHandling";
      InverterDriveProcessing_DB : "InverterDriveProcessing";
      DigitalInputProcessing_DB { ExternalAccessible := 'False'; ExternalVisible := 'False'; ExternalWritable := 'False'} : "DigitalInputProcessing";
      Simulation_DB { ExternalAccessible := 'False'; ExternalVisible := 'False'; ExternalWritable := 'False'} : "Simulation";
      HBL_HV_640 { S7_SetPoint := 'True'} : "fbProcessValve2_V2";
      HBL_HV_670 { S7_SetPoint := 'True'} : "fbProcessValve2_V2";
      CPC_HV_852 { S7_SetPoint := 'True'} : "fbProcessValve2_V2";
      HBL_HV_861 { S7_SetPoint := 'True'} : "fbProcessValve2_V2";
      bTempOpenReq { S7_SetPoint := 'True'} : Bool;
      bTempCloseReq : Bool;
      bTempOpenStat : Bool;
      bTempCloseStat : Bool;
   END_VAR
BEGIN

REGION Network 1: Digital inputs
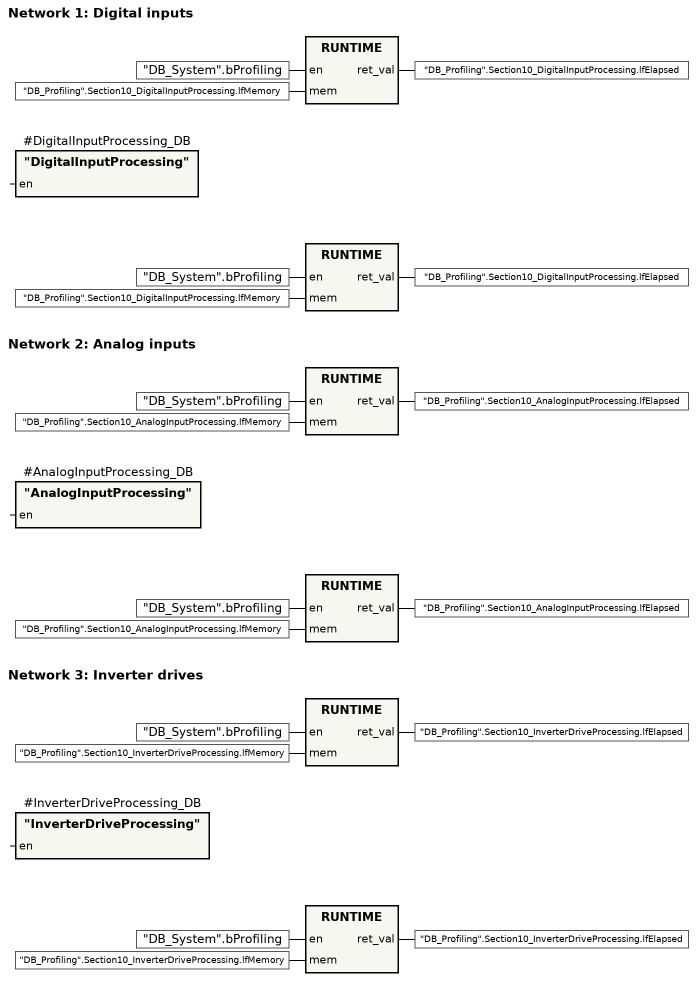
   // no SCL statement known for Runtime: written as a call
   IF "DB_System".bProfiling THEN
       "DB_Profiling".Section10_DigitalInputProcessing.lfElapsed := Runtime(mem := "DB_Profiling".Section10_DigitalInputProcessing.lfMemory);
   END_IF;
   #DigitalInputProcessing_DB();   // "DigitalInputProcessing"
   IF "DB_System".bProfiling THEN
       "DB_Profiling".Section10_DigitalInputProcessing.lfElapsed := Runtime(mem := "DB_Profiling".Section10_DigitalInputProcessing.lfMemory);
   END_IF;
END_REGION

REGION Network 2: Analog inputs
   // no SCL statement known for Runtime: written as a call
   IF "DB_System".bProfiling THEN
       "DB_Profiling".Section10_AnalogInputProcessing.lfElapsed := Runtime(mem := "DB_Profiling".Section10_AnalogInputProcessing.lfMemory);
   END_IF;
   #AnalogInputProcessing_DB();   // "AnalogInputProcessing"
   IF "DB_System".bProfiling THEN
       "DB_Profiling".Section10_AnalogInputProcessing.lfElapsed := Runtime(mem := "DB_Profiling".Section10_AnalogInputProcessing.lfMemory);
   END_IF;
END_REGION

REGION Network 3: Inverter drives
   // no SCL statement known for Runtime: written as a call
   IF "DB_System".bProfiling THEN
       "DB_Profiling".Section10_InverterDriveProcessing.lfElapsed := Runtime(mem := "DB_Profiling".Section10_InverterDriveProcessing.lfMemory);
   END_IF;
   #InverterDriveProcessing_DB();   // "InverterDriveProcessing"
   IF "DB_System".bProfiling THEN
       "DB_Profiling".Section10_InverterDriveProcessing.lfElapsed := Runtime(mem := "DB_Profiling".Section10_InverterDriveProcessing.lfMemory);
   END_IF;
END_REGION

REGION Network 4: Process valves
   // Own FB?
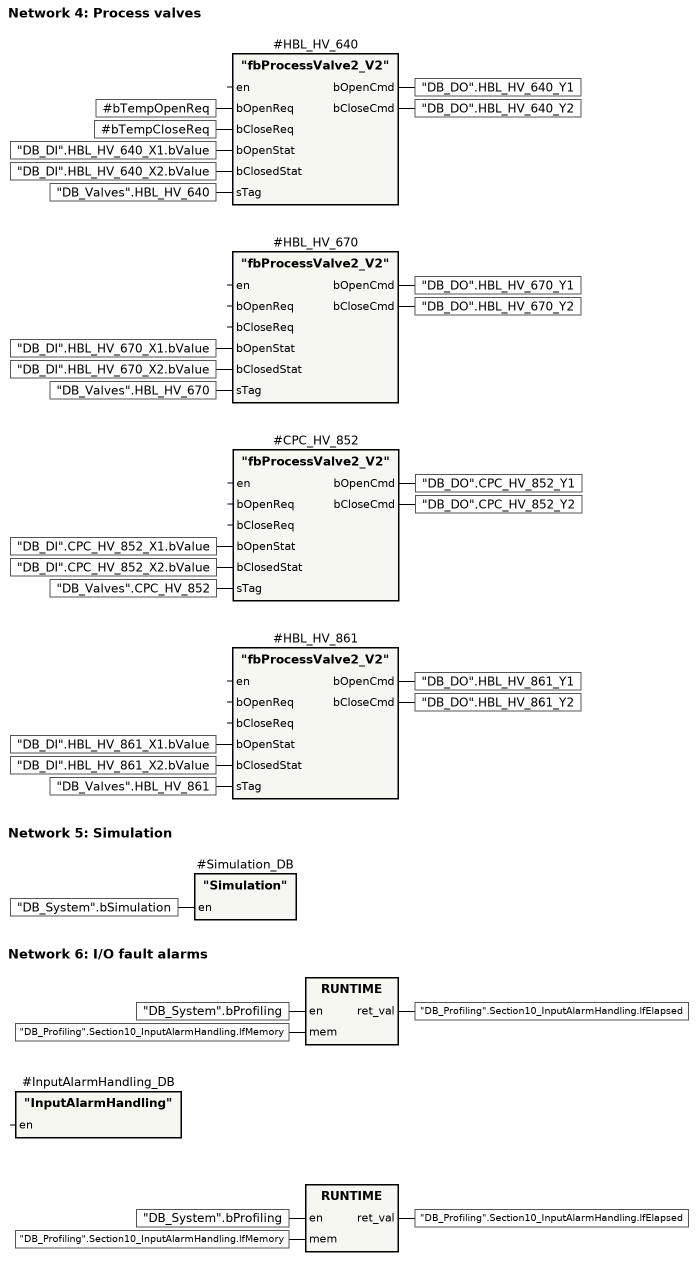
   #HBL_HV_640(bOpenReq := #bTempOpenReq,   // "fbProcessValve2_V2"
               bCloseReq := #bTempCloseReq,
               bOpenStat := "DB_DI".HBL_HV_640_X1.bValue,
               bClosedStat := "DB_DI".HBL_HV_640_X2.bValue,
               sTag := "DB_Valves".HBL_HV_640,
               bOpenCmd => "DB_DO".HBL_HV_640_Y1,
               bCloseCmd => "DB_DO".HBL_HV_640_Y2);
   #HBL_HV_670(bOpenStat := "DB_DI".HBL_HV_670_X1.bValue,   // "fbProcessValve2_V2"
               bClosedStat := "DB_DI".HBL_HV_670_X2.bValue,
               sTag := "DB_Valves".HBL_HV_670,
               bOpenCmd => "DB_DO".HBL_HV_670_Y1,
               bCloseCmd => "DB_DO".HBL_HV_670_Y2);
   #CPC_HV_852(bOpenStat := "DB_DI".CPC_HV_852_X1.bValue,   // "fbProcessValve2_V2"
               bClosedStat := "DB_DI".CPC_HV_852_X2.bValue,
               sTag := "DB_Valves".CPC_HV_852,
               bOpenCmd => "DB_DO".CPC_HV_852_Y1,
               bCloseCmd => "DB_DO".CPC_HV_852_Y2);
   #HBL_HV_861(bOpenStat := "DB_DI".HBL_HV_861_X1.bValue,   // "fbProcessValve2_V2"
               bClosedStat := "DB_DI".HBL_HV_861_X2.bValue,
               sTag := "DB_Valves".HBL_HV_861,
               bOpenCmd => "DB_DO".HBL_HV_861_Y1,
               bCloseCmd => "DB_DO".HBL_HV_861_Y2);
END_REGION

REGION Network 5: Simulation
   IF "DB_System".bSimulation THEN
       #Simulation_DB();   // "Simulation"
   END_IF;
END_REGION

REGION Network 6: I/O fault alarms
   // Put this last so that any Simulation code doesn't have to fix up any alarms
   // no SCL statement known for Runtime: written as a call
   IF "DB_System".bProfiling THEN
       "DB_Profiling".Section10_InputAlarmHandling.lfElapsed := Runtime(mem := "DB_Profiling".Section10_InputAlarmHandling.lfMemory);
   END_IF;
   #InputAlarmHandling_DB();   // "InputAlarmHandling"
   IF "DB_System".bProfiling THEN
       "DB_Profiling".Section10_InputAlarmHandling.lfElapsed := Runtime(mem := "DB_Profiling".Section10_InputAlarmHandling.lfMemory);
   END_IF;
END_REGION
END_FUNCTION_BLOCK

FUNCTION_BLOCK "DigitalInputProcessing"   // FB8, FBD
TITLE = Handle digital input signals
{ S7_Optimized_Access := 'TRUE' }
AUTHOR : Heaten
VERSION : 0.1
// Map, validate and process digital inputs
// stored: AutoNumber true, IsIECCheckEnabled false, IsRetainMemResEnabled false, MemoryReserve 0, SetENOAutomatically false, UDAEnableTagReadback false
   VAR
      HBL_LS_632 { ExternalAccessible := 'False'; ExternalVisible := 'False'; ExternalWritable := 'False'} : "stAnalogInput";
      HBL_LS_633 { S7_SetPoint := 'True'} : "stAnalogInput";
      HBL_LS_644 { S7_SetPoint := 'True'} : "stAnalogInput";
      HBL_LS_674 { S7_SetPoint := 'True'} : "stAnalogInput";
      Dummy { ExternalAccessible := 'False'; ExternalVisible := 'False'; ExternalWritable := 'False'} : Bool;
      LS632 : Real;
      LS633 : Real;
      LS644 : Real;
      LS674 : Real;
   END_VAR
   // HBL_LS_632.Raw.iMin := 0;
   // HBL_LS_632.Raw.iMax := 27648;
   // HBL_LS_632.Eng.fMin := 4.0;   // [mA]
   // HBL_LS_632.Eng.fMax := 20.0;   // [mA]
   // HBL_LS_633.Raw.iMin := 0;
   // HBL_LS_633.Raw.iMax := 27648;
   // HBL_LS_633.Eng.fMin := 4.0;   // [mA]
   // HBL_LS_633.Eng.fMax := 20.0;   // [mA]
   // HBL_LS_644.Eng.fMin := 4.0;
   // HBL_LS_644.Eng.fMax := 20.0;
   // HBL_LS_674.Eng.fMin := 4.0;
   // HBL_LS_674.Eng.fMax := 20.0;
BEGIN

REGION Network 1: Emergency stop status
   // Polarity of input is preserved. 1 = No E-stop, 0 = E-stop
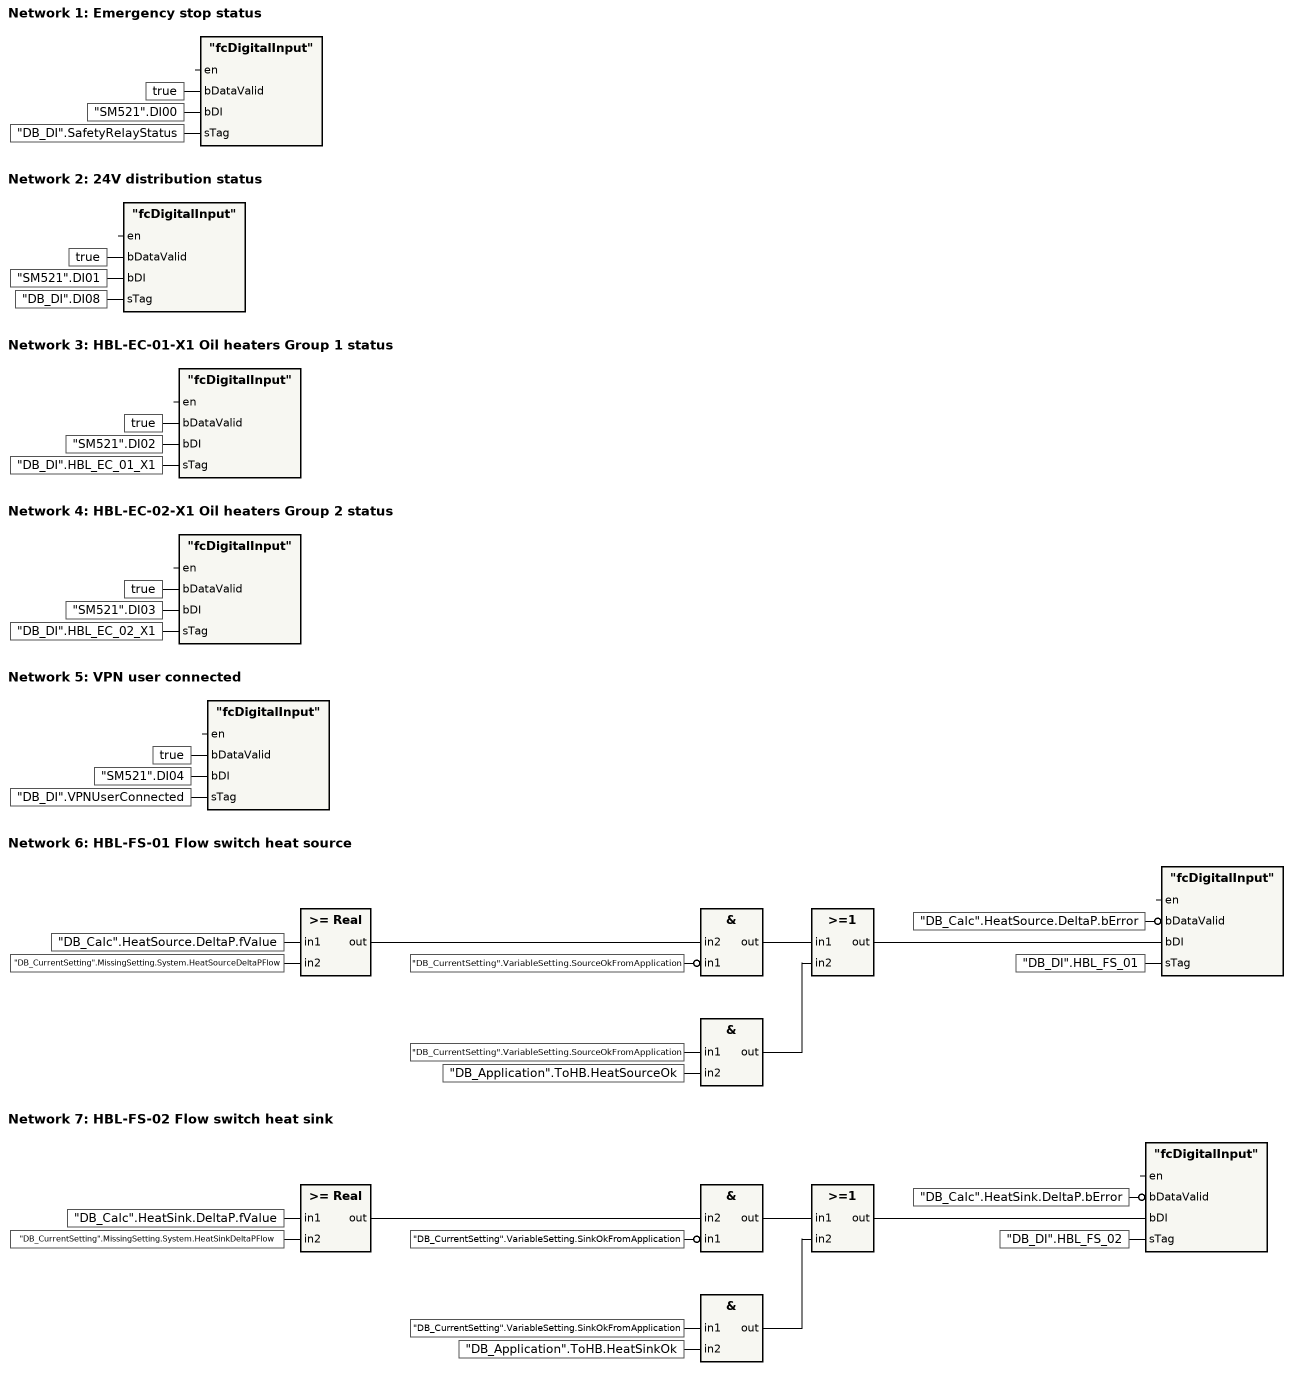
   "fcDigitalInput"(bDataValid := true, bDI := "SM521".DI00, sTag := "DB_DI".SafetyRelayStatus);
END_REGION

REGION Network 2: 24V distribution status
   "fcDigitalInput"(bDataValid := true, bDI := "SM521".DI01, sTag := "DB_DI".DI08);
END_REGION

REGION Network 3: HBL-EC-01-X1 Oil heaters Group 1 status
   "fcDigitalInput"(bDataValid := true, bDI := "SM521".DI02, sTag := "DB_DI".HBL_EC_01_X1);
END_REGION

REGION Network 4: HBL-EC-02-X1 Oil heaters Group 2 status
   "fcDigitalInput"(bDataValid := true, bDI := "SM521".DI03, sTag := "DB_DI".HBL_EC_02_X1);
END_REGION

REGION Network 5: VPN user connected
   "fcDigitalInput"(bDataValid := true, bDI := "SM521".DI04, sTag := "DB_DI".VPNUserConnected);
END_REGION

REGION Network 6: HBL-FS-01 Flow switch heat source
   // Virtual instrument:
   //  - Generate this locally from the pressure difference across the evaporator
   //  - Let the Application PLC do it based on input from the host process
   "fcDigitalInput"(bDataValid := NOT "DB_Calc".HeatSource.DeltaP.bError,
                    bDI := (("DB_Calc".HeatSource.DeltaP.fValue >= "DB_CurrentSetting".MissingSetting.System.HeatSourceDeltaPFlow) AND NOT "DB_CurrentSetting".VariableSetting.SourceOkFromApplication) OR ("DB_CurrentSetting".VariableSetting.SourceOkFromApplication AND "DB_Application".ToHB.HeatSourceOk),
                    sTag := "DB_DI".HBL_FS_01);
END_REGION

REGION Network 7: HBL-FS-02 Flow switch heat sink
   // Virtual instrument:
   //  - Generate this from the pressure difference across the condenser
   //  - Let the Application PLC does it based on input from the host process
   "fcDigitalInput"(bDataValid := NOT "DB_Calc".HeatSink.DeltaP.bError,
                    bDI := (("DB_Calc".HeatSink.DeltaP.fValue >= "DB_CurrentSetting".MissingSetting.System.HeatSinkDeltaPFlow) AND NOT "DB_CurrentSetting".VariableSetting.SinkOkFromApplication) OR ("DB_CurrentSetting".VariableSetting.SinkOkFromApplication AND "DB_Application".ToHB.HeatSinkOk),
                    sTag := "DB_DI".HBL_FS_02);
END_REGION

REGION Network 8: HBL-PS-500-X2 Compressor discharge overpressure
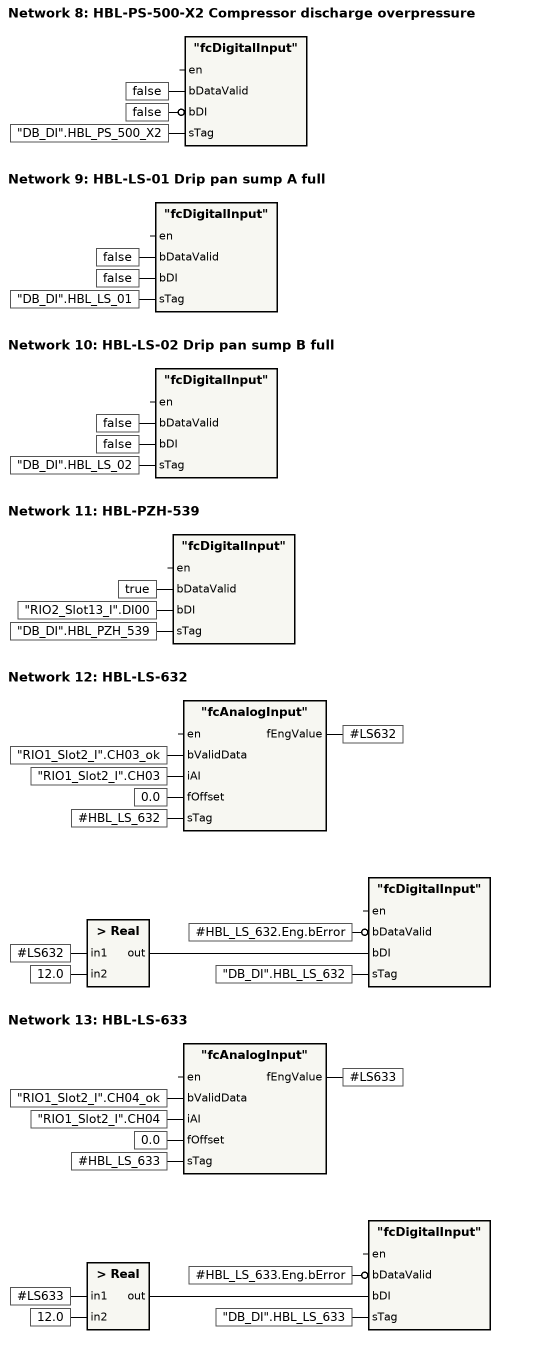
   "fcDigitalInput"(bDataValid := false, bDI := NOT false, sTag := "DB_DI".HBL_PS_500_X2);
END_REGION

REGION Network 9: HBL-LS-01 Drip pan sump A full
   "fcDigitalInput"(bDataValid := false, bDI := false, sTag := "DB_DI".HBL_LS_01);
END_REGION

REGION Network 10: HBL-LS-02 Drip pan sump B full
   "fcDigitalInput"(bDataValid := false, bDI := false, sTag := "DB_DI".HBL_LS_02);
END_REGION

REGION Network 11: HBL-PZH-539
   "fcDigitalInput"(bDataValid := true, bDI := "RIO2_Slot13_I".DI00, sTag := "DB_DI".HBL_PZH_539);
END_REGION

REGION Network 12: HBL-LS-632
   // 2-wire level switch. Low = 8mA, High = 16mA. Use a 12mA threshold to switch HI/LO
   "fcAnalogInput"(bValidData := "RIO1_Slot2_I".CH03_ok,
                   iAI := "RIO1_Slot2_I".CH03,
                   fOffset := 0.0,
                   sTag := #HBL_LS_632,
                   fEngValue => #LS632);
   "fcDigitalInput"(bDataValid := NOT #HBL_LS_632.Eng.bError, bDI := #LS632 > 12.0, sTag := "DB_DI".HBL_LS_632);
END_REGION

REGION Network 13: HBL-LS-633
   // 2-wire level switch. Low = 8mA, High = 16mA. Use a 12mA threshold to switch HI/LO
   "fcAnalogInput"(bValidData := "RIO1_Slot2_I".CH04_ok,
                   iAI := "RIO1_Slot2_I".CH04,
                   fOffset := 0.0,
                   sTag := #HBL_LS_633,
                   fEngValue => #LS633);
   "fcDigitalInput"(bDataValid := NOT #HBL_LS_633.Eng.bError, bDI := #LS633 > 12.0, sTag := "DB_DI".HBL_LS_633);
END_REGION

REGION Network 14: HBL-LS-644
   // 2-wire level switch. Low = 8mA, High = 16mA. Use a 12mA threshold to switch HI/LO
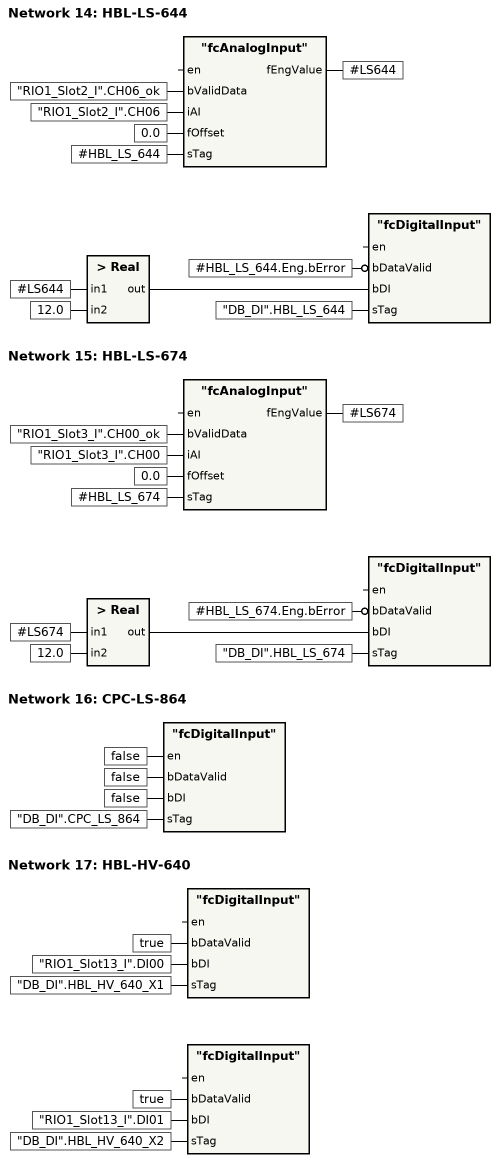
   "fcAnalogInput"(bValidData := "RIO1_Slot2_I".CH06_ok,
                   iAI := "RIO1_Slot2_I".CH06,
                   fOffset := 0.0,
                   sTag := #HBL_LS_644,
                   fEngValue => #LS644);
   "fcDigitalInput"(bDataValid := NOT #HBL_LS_644.Eng.bError, bDI := #LS644 > 12.0, sTag := "DB_DI".HBL_LS_644);
END_REGION

REGION Network 15: HBL-LS-674
   // 2-wire level switch. Low = 8mA, High = 16mA. Use a 12mA threshold to switch HI/LO
   "fcAnalogInput"(bValidData := "RIO1_Slot3_I".CH00_ok,
                   iAI := "RIO1_Slot3_I".CH00,
                   fOffset := 0.0,
                   sTag := #HBL_LS_674,
                   fEngValue => #LS674);
   "fcDigitalInput"(bDataValid := NOT #HBL_LS_674.Eng.bError, bDI := #LS674 > 12.0, sTag := "DB_DI".HBL_LS_674);
END_REGION

REGION Network 16: CPC-LS-864
   IF false THEN "fcDigitalInput"(bDataValid := false, bDI := false, sTag := "DB_DI".CPC_LS_864); END_IF;
END_REGION

REGION Network 17: HBL-HV-640
   "fcDigitalInput"(bDataValid := true, bDI := "RIO1_Slot13_I".DI00, sTag := "DB_DI".HBL_HV_640_X1);
   "fcDigitalInput"(bDataValid := true, bDI := "RIO1_Slot13_I".DI01, sTag := "DB_DI".HBL_HV_640_X2);
END_REGION

REGION Network 18: HBL-HV-670
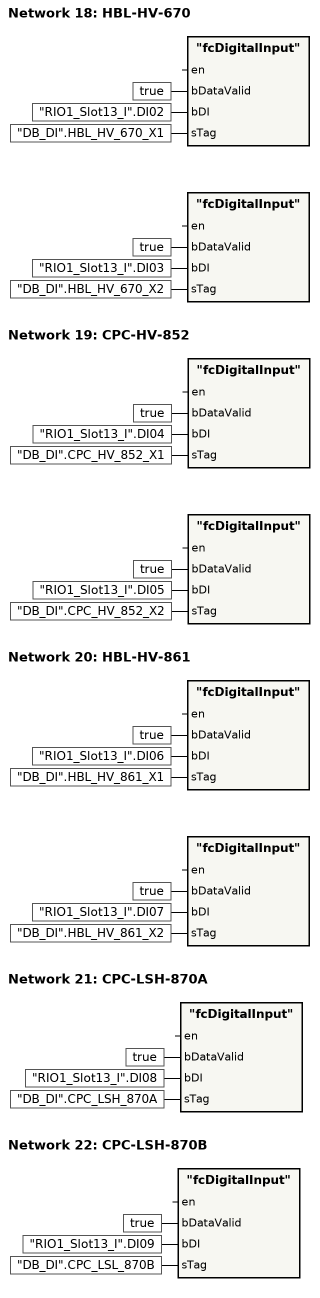
   "fcDigitalInput"(bDataValid := true, bDI := "RIO1_Slot13_I".DI02, sTag := "DB_DI".HBL_HV_670_X1);
   "fcDigitalInput"(bDataValid := true, bDI := "RIO1_Slot13_I".DI03, sTag := "DB_DI".HBL_HV_670_X2);
END_REGION

REGION Network 19: CPC-HV-852
   // '
   "fcDigitalInput"(bDataValid := true, bDI := "RIO1_Slot13_I".DI04, sTag := "DB_DI".CPC_HV_852_X1);
   "fcDigitalInput"(bDataValid := true, bDI := "RIO1_Slot13_I".DI05, sTag := "DB_DI".CPC_HV_852_X2);
END_REGION

REGION Network 20: HBL-HV-861
   // '
   "fcDigitalInput"(bDataValid := true, bDI := "RIO1_Slot13_I".DI06, sTag := "DB_DI".HBL_HV_861_X1);
   "fcDigitalInput"(bDataValid := true, bDI := "RIO1_Slot13_I".DI07, sTag := "DB_DI".HBL_HV_861_X2);
END_REGION

REGION Network 21: CPC-LSH-870A
   "fcDigitalInput"(bDataValid := true, bDI := "RIO1_Slot13_I".DI08, sTag := "DB_DI".CPC_LSH_870A);
END_REGION

REGION Network 22: CPC-LSH-870B
   "fcDigitalInput"(bDataValid := true, bDI := "RIO1_Slot13_I".DI09, sTag := "DB_DI".CPC_LSL_870B);
END_REGION

REGION Network 23: CPC-PZH-874
